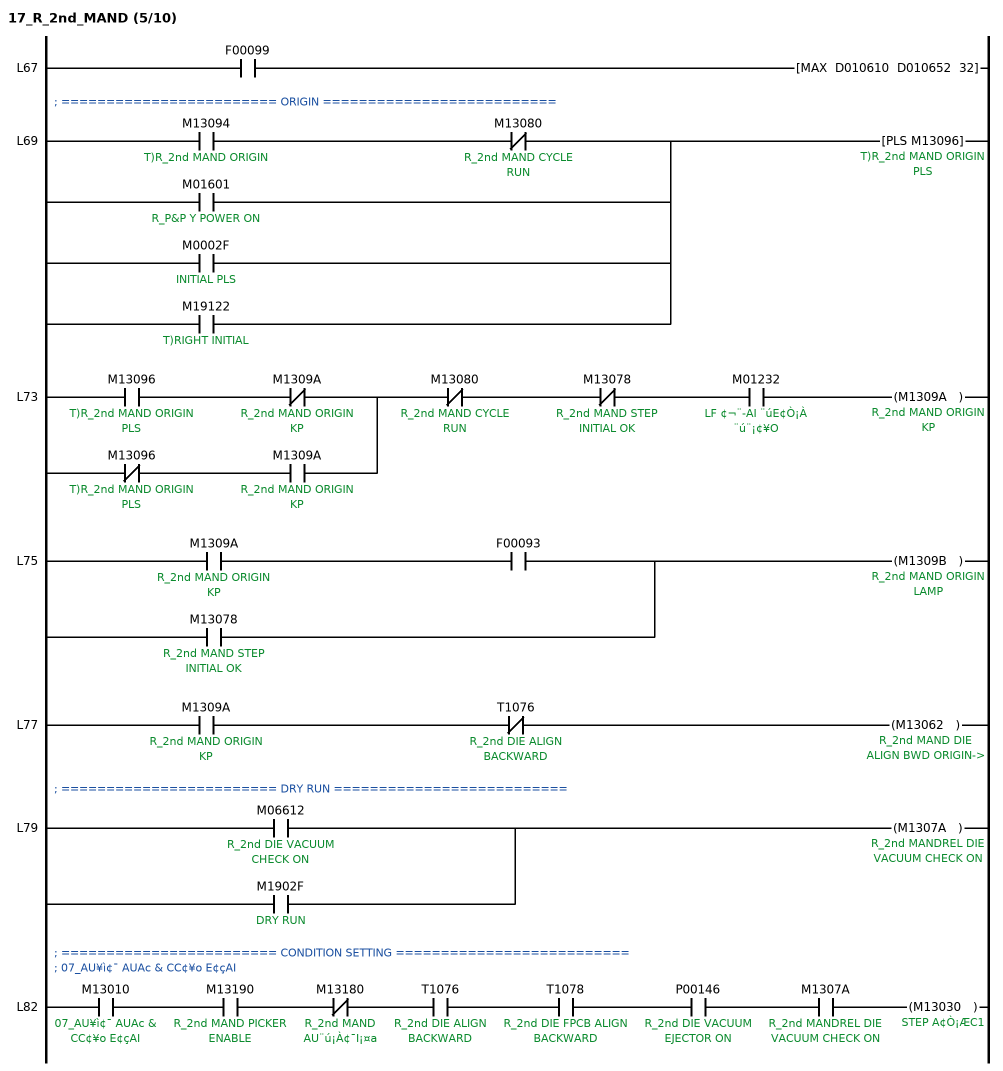
[picture p144: 17_R_2nd_MAND rungs L67-L82]
; L67
LOAD      F00099
MAX       D010610 D010652 32
// ======================== ORIGIN ==========================
; L69
LOAD      M13094	// T)R_2nd MAND ORIGIN
AND NOT   M13080	// R_2nd MAND CYCLE RUN
OR        M01601	// R_P&P Y POWER ON
OR        M0002F	// INITIAL PLS
OR        M19122	// T)RIGHT INITIAL
OUTP      M13096	// T)R_2nd MAND ORIGIN PLS
; L73
LOAD      M13096	// T)R_2nd MAND ORIGIN PLS
AND NOT   M1309A	// R_2nd MAND ORIGIN KP
LOAD NOT  M13096	// T)R_2nd MAND ORIGIN PLS
AND       M1309A	// R_2nd MAND ORIGIN KP
OR LOAD
AND NOT   M13080	// R_2nd MAND CYCLE RUN
AND NOT   M13078	// R_2nd MAND STEP INITIAL OK
AND       M01232	// LF ¢¬¨­AI ¨úE¢Ò¡À ¨ú¨¡¢¥O
OUT       M1309A	// R_2nd MAND ORIGIN KP
; L75
LOAD      M1309A	// R_2nd MAND ORIGIN KP
AND       F00093
OR        M13078	// R_2nd MAND STEP INITIAL OK
OUT       M1309B	// R_2nd MAND ORIGIN LAMP
; L77
LOAD      M1309A	// R_2nd MAND ORIGIN KP
AND NOT   T1076	// R_2nd DIE ALIGN BACKWARD
OUT       M13062	// R_2nd MAND DIE ALIGN BWD ORIGIN->
// ======================== DRY RUN ==========================
; L79
LOAD      M06612	// R_2nd DIE VACUUM CHECK ON
OR        M1902F	// DRY RUN
OUT       M1307A	// R_2nd MANDREL DIE VACUUM CHECK ON
// ======================== CONDITION SETTING ==========================
; L82
LOAD      M13010	// 07_AU¥ì¢¯ AUAc & CC¢¥o E¢çAI
AND       M13190	// R_2nd MAND PICKER ENABLE
AND NOT   M13180	// R_2nd MAND AU¨ú¡À¢¯I¡¤a
AND       T1076	// R_2nd DIE ALIGN BACKWARD
AND       T1078	// R_2nd DIE FPCB ALIGN BACKWARD
AND       P00146	// R_2nd DIE VACUUM EJECTOR ON
AND       M1307A	// R_2nd MANDREL DIE VACUUM CHECK ON
OUT       M13030	// STEP A¢Ò¡ÆC1
// output comment: 07_AU¥ì¢¯ AUAc & CC¢¥o E¢çAI

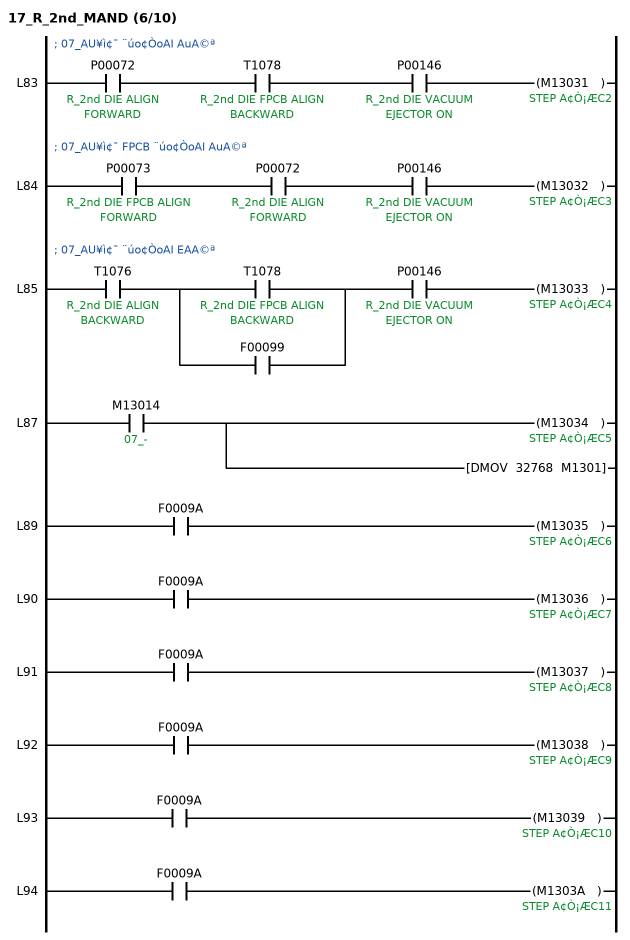
; L83
LOAD      P00072	// R_2nd DIE ALIGN FORWARD
AND       T1078	// R_2nd DIE FPCB ALIGN BACKWARD
AND       P00146	// R_2nd DIE VACUUM EJECTOR ON
OUT       M13031	// STEP A¢Ò¡ÆC2
// output comment: 07_AU¥ì¢¯ ¨úo¢ÒoAI AuA©ª
; L84
LOAD      P00073	// R_2nd DIE FPCB ALIGN FORWARD
AND       P00072	// R_2nd DIE ALIGN FORWARD
AND       P00146	// R_2nd DIE VACUUM EJECTOR ON
OUT       M13032	// STEP A¢Ò¡ÆC3
// output comment: 07_AU¥ì¢¯ FPCB ¨úo¢ÒoAI AuA©ª
; L85
LOAD      T1076	// R_2nd DIE ALIGN BACKWARD
LOAD      T1078	// R_2nd DIE FPCB ALIGN BACKWARD
OR        F00099
AND LOAD
AND       P00146	// R_2nd DIE VACUUM EJECTOR ON
OUT       M13033	// STEP A¢Ò¡ÆC4
// output comment: 07_AU¥ì¢¯ ¨úo¢ÒoAI EAA©ª
; L87
LOAD      M13014	// 07_-
OUT       M13034	// STEP A¢Ò¡ÆC5
DMOV      32768 M1301
; L89
LOAD      F0009A
OUT       M13035	// STEP A¢Ò¡ÆC6
; L90
LOAD      F0009A
OUT       M13036	// STEP A¢Ò¡ÆC7
; L91
LOAD      F0009A
OUT       M13037	// STEP A¢Ò¡ÆC8
; L92
LOAD      F0009A
OUT       M13038	// STEP A¢Ò¡ÆC9
; L93
LOAD      F0009A
OUT       M13039	// STEP A¢Ò¡ÆC10
; L94
LOAD      F0009A
OUT       M1303A	// STEP A¢Ò¡ÆC11

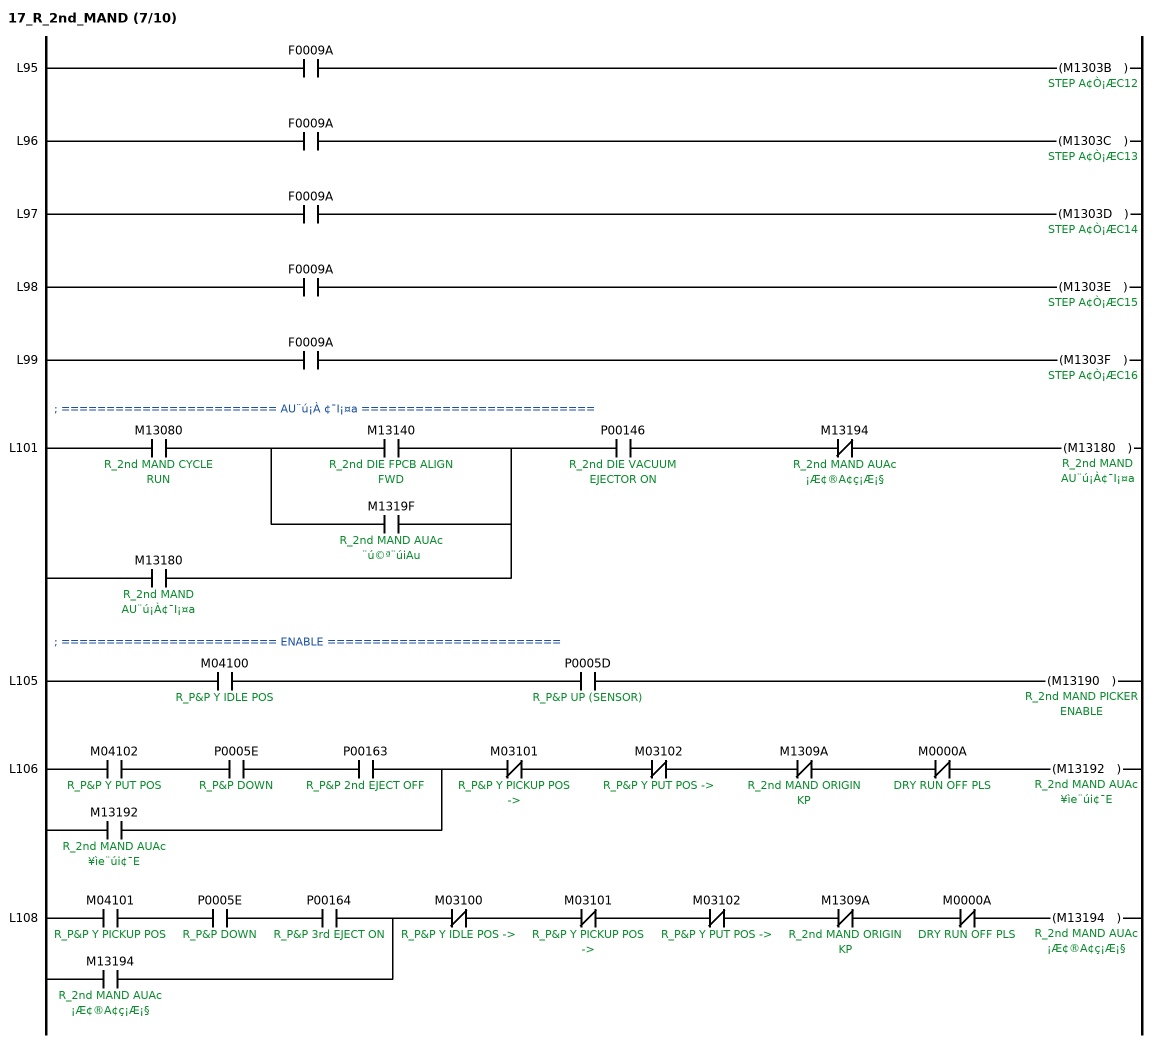
; L95
LOAD      F0009A
OUT       M1303B	// STEP A¢Ò¡ÆC12
; L96
LOAD      F0009A
OUT       M1303C	// STEP A¢Ò¡ÆC13
; L97
LOAD      F0009A
OUT       M1303D	// STEP A¢Ò¡ÆC14
; L98
LOAD      F0009A
OUT       M1303E	// STEP A¢Ò¡ÆC15
; L99
LOAD      F0009A
OUT       M1303F	// STEP A¢Ò¡ÆC16
// ======================== AU¨ú¡À ¢¯I¡¤a ==========================
; L101
LOAD      M13080	// R_2nd MAND CYCLE RUN
LOAD      M13140	// R_2nd DIE FPCB ALIGN FWD
OR        M1319F	// R_2nd MAND AUAc ¨ú©ª¨úiAu
AND LOAD
OR        M13180	// R_2nd MAND AU¨ú¡À¢¯I¡¤a
AND       P00146	// R_2nd DIE VACUUM EJECTOR ON
AND NOT   M13194	// R_2nd MAND AUAc ¡Æ¢®A¢ç¡Æ¡§
OUT       M13180	// R_2nd MAND AU¨ú¡À¢¯I¡¤a
// ======================== ENABLE ==========================
; L105
LOAD      M04100	// R_P&P Y IDLE POS
AND       P0005D	// R_P&P UP (SENSOR)
OUT       M13190	// R_2nd MAND PICKER ENABLE
; L106
LOAD      M04102	// R_P&P Y PUT POS
AND       P0005E	// R_P&P DOWN
AND       P00163	// R_P&P 2nd EJECT OFF
OR        M13192	// R_2nd MAND AUAc ¥ìe¨úi¢¯E
AND NOT   M03101	// R_P&P Y PICKUP POS ->
AND NOT   M03102	// R_P&P Y PUT POS ->
AND NOT   M1309A	// R_2nd MAND ORIGIN KP
AND NOT   M0000A	// DRY RUN OFF PLS
OUT       M13192	// R_2nd MAND AUAc ¥ìe¨úi¢¯E
; L108
LOAD      M04101	// R_P&P Y PICKUP POS
AND       P0005E	// R_P&P DOWN
AND       P00164	// R_P&P 3rd EJECT ON
OR        M13194	// R_2nd MAND AUAc ¡Æ¢®A¢ç¡Æ¡§
AND NOT   M03100	// R_P&P Y IDLE POS ->
AND NOT   M03101	// R_P&P Y PICKUP POS ->
AND NOT   M03102	// R_P&P Y PUT POS ->
AND NOT   M1309A	// R_2nd MAND ORIGIN KP
AND NOT   M0000A	// DRY RUN OFF PLS
OUT       M13194	// R_2nd MAND AUAc ¡Æ¢®A¢ç¡Æ¡§

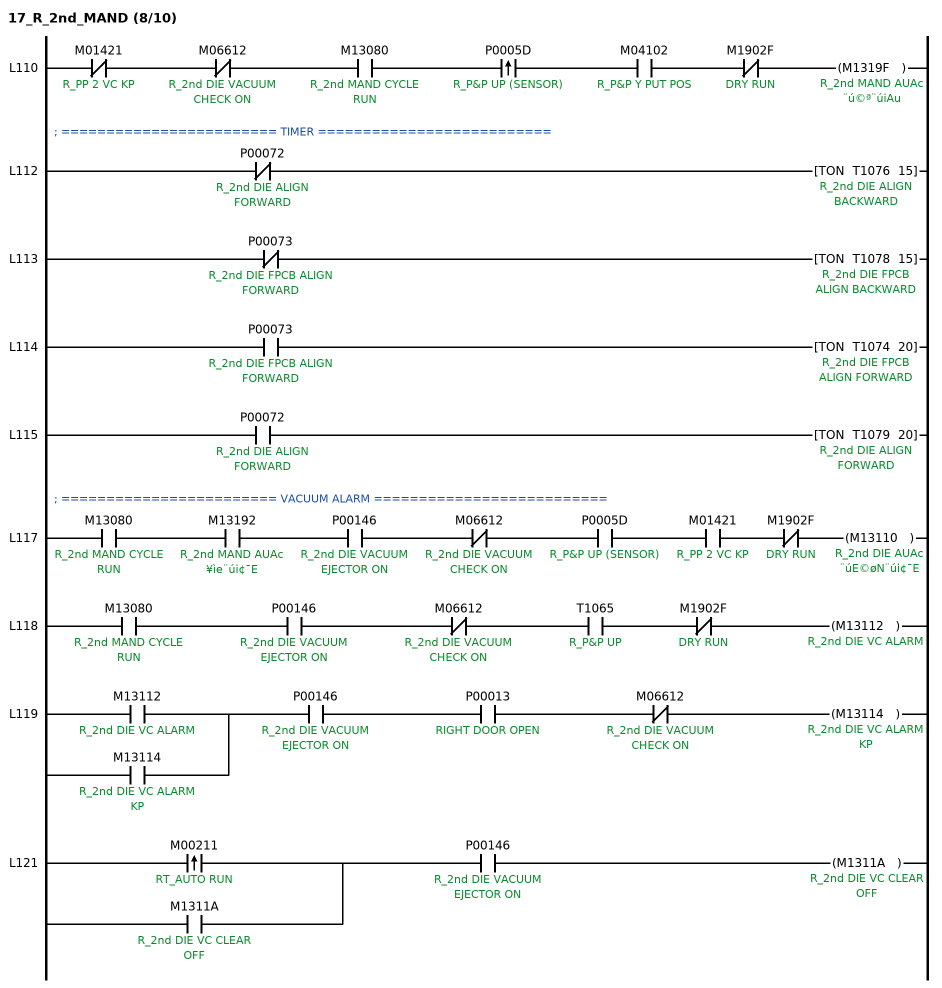
; L110
LOAD NOT  M01421	// R_PP 2 VC KP
AND NOT   M06612	// R_2nd DIE VACUUM CHECK ON
AND       M13080	// R_2nd MAND CYCLE RUN
ANDP      P0005D	// R_P&P UP (SENSOR)
AND       M04102	// R_P&P Y PUT POS
AND NOT   M1902F	// DRY RUN
OUT       M1319F	// R_2nd MAND AUAc ¨ú©ª¨úiAu
// ======================== TIMER ==========================
; L112
LOAD NOT  P00072	// R_2nd DIE ALIGN FORWARD
TON       T1076 15	// R_2nd DIE ALIGN BACKWARD
; L113
LOAD NOT  P00073	// R_2nd DIE FPCB ALIGN FORWARD
TON       T1078 15	// R_2nd DIE FPCB ALIGN BACKWARD
; L114
LOAD      P00073	// R_2nd DIE FPCB ALIGN FORWARD
TON       T1074 20	// R_2nd DIE FPCB ALIGN FORWARD
; L115
LOAD      P00072	// R_2nd DIE ALIGN FORWARD
TON       T1079 20	// R_2nd DIE ALIGN FORWARD
// ======================== VACUUM ALARM ==========================
; L117
LOAD      M13080	// R_2nd MAND CYCLE RUN
AND       M13192	// R_2nd MAND AUAc ¥ìe¨úi¢¯E
AND       P00146	// R_2nd DIE VACUUM EJECTOR ON
AND NOT   M06612	// R_2nd DIE VACUUM CHECK ON
AND       P0005D	// R_P&P UP (SENSOR)
AND       M01421	// R_PP 2 VC KP
AND NOT   M1902F	// DRY RUN
OUT       M13110	// R_2nd DIE AUAc ¨úE©øN¨úi¢¯E
; L118
LOAD      M13080	// R_2nd MAND CYCLE RUN
AND       P00146	// R_2nd DIE VACUUM EJECTOR ON
AND NOT   M06612	// R_2nd DIE VACUUM CHECK ON
AND       T1065	// R_P&P UP
AND NOT   M1902F	// DRY RUN
OUT       M13112	// R_2nd DIE VC ALARM
; L119
LOAD      M13112	// R_2nd DIE VC ALARM
OR        M13114	// R_2nd DIE VC ALARM KP
AND       P00146	// R_2nd DIE VACUUM EJECTOR ON
AND       P00013	// RIGHT DOOR OPEN
AND NOT   M06612	// R_2nd DIE VACUUM CHECK ON
OUT       M13114	// R_2nd DIE VC ALARM KP
; L121
LOADP     M00211	// RT_AUTO RUN
OR        M1311A	// R_2nd DIE VC CLEAR OFF
AND       P00146	// R_2nd DIE VACUUM EJECTOR ON
OUT       M1311A	// R_2nd DIE VC CLEAR OFF

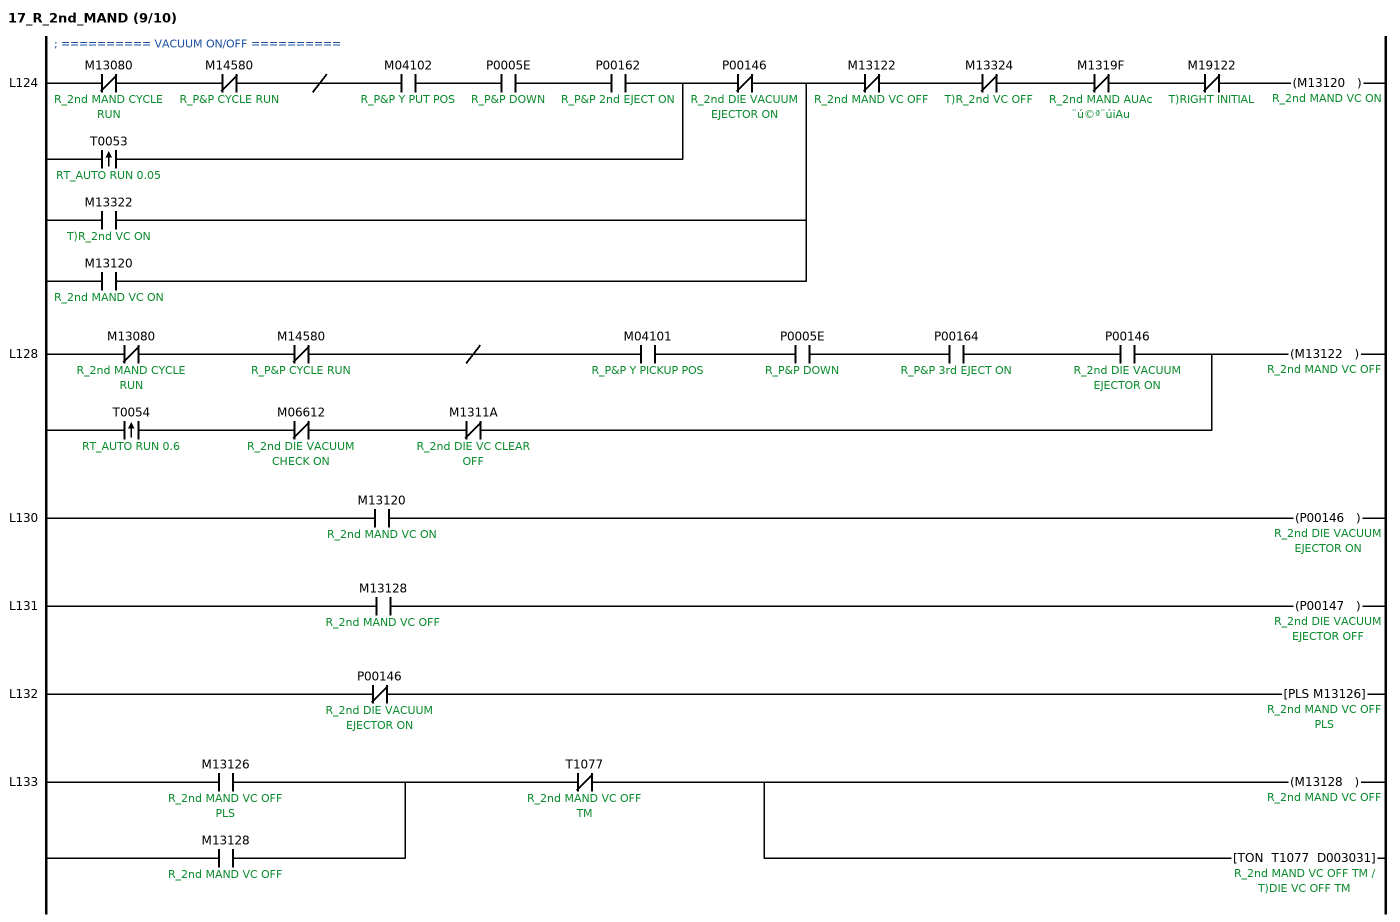
// ========== VACUUM ON/OFF ==========
; L124
LOAD NOT  M13080	// R_2nd MAND CYCLE RUN
AND NOT   M14580	// R_P&P CYCLE RUN
NOT
AND       M04102	// R_P&P Y PUT POS
AND       P0005E	// R_P&P DOWN
AND       P00162	// R_P&P 2nd EJECT ON
ORP       T0053	// RT_AUTO RUN 0.05
AND NOT   P00146	// R_2nd DIE VACUUM EJECTOR ON
OR        M13322	// T)R_2nd VC ON
OR        M13120	// R_2nd MAND VC ON
AND NOT   M13122	// R_2nd MAND VC OFF
AND NOT   M13324	// T)R_2nd VC OFF
AND NOT   M1319F	// R_2nd MAND AUAc ¨ú©ª¨úiAu
AND NOT   M19122	// T)RIGHT INITIAL
OUT       M13120	// R_2nd MAND VC ON
; L128
LOAD NOT  M13080	// R_2nd MAND CYCLE RUN
AND NOT   M14580	// R_P&P CYCLE RUN
NOT
AND       M04101	// R_P&P Y PICKUP POS
AND       P0005E	// R_P&P DOWN
AND       P00164	// R_P&P 3rd EJECT ON
AND       P00146	// R_2nd DIE VACUUM EJECTOR ON
LOADP     T0054	// RT_AUTO RUN 0.6
AND NOT   M06612	// R_2nd DIE VACUUM CHECK ON
AND NOT   M1311A	// R_2nd DIE VC CLEAR OFF
OR LOAD
OUT       M13122	// R_2nd MAND VC OFF
; L130
LOAD      M13120	// R_2nd MAND VC ON
OUT       P00146	// R_2nd DIE VACUUM EJECTOR ON
; L131
LOAD      M13128	// R_2nd MAND VC OFF
OUT       P00147	// R_2nd DIE VACUUM EJECTOR OFF
; L132
LOAD NOT  P00146	// R_2nd DIE VACUUM EJECTOR ON
OUTP      M13126	// R_2nd MAND VC OFF PLS
; L133
LOAD      M13126	// R_2nd MAND VC OFF PLS
OR        M13128	// R_2nd MAND VC OFF
AND NOT   T1077	// R_2nd MAND VC OFF TM
OUT       M13128	// R_2nd MAND VC OFF
TON       T1077 D003031	// R_2nd MAND VC OFF TM / T)DIE VC OFF TM

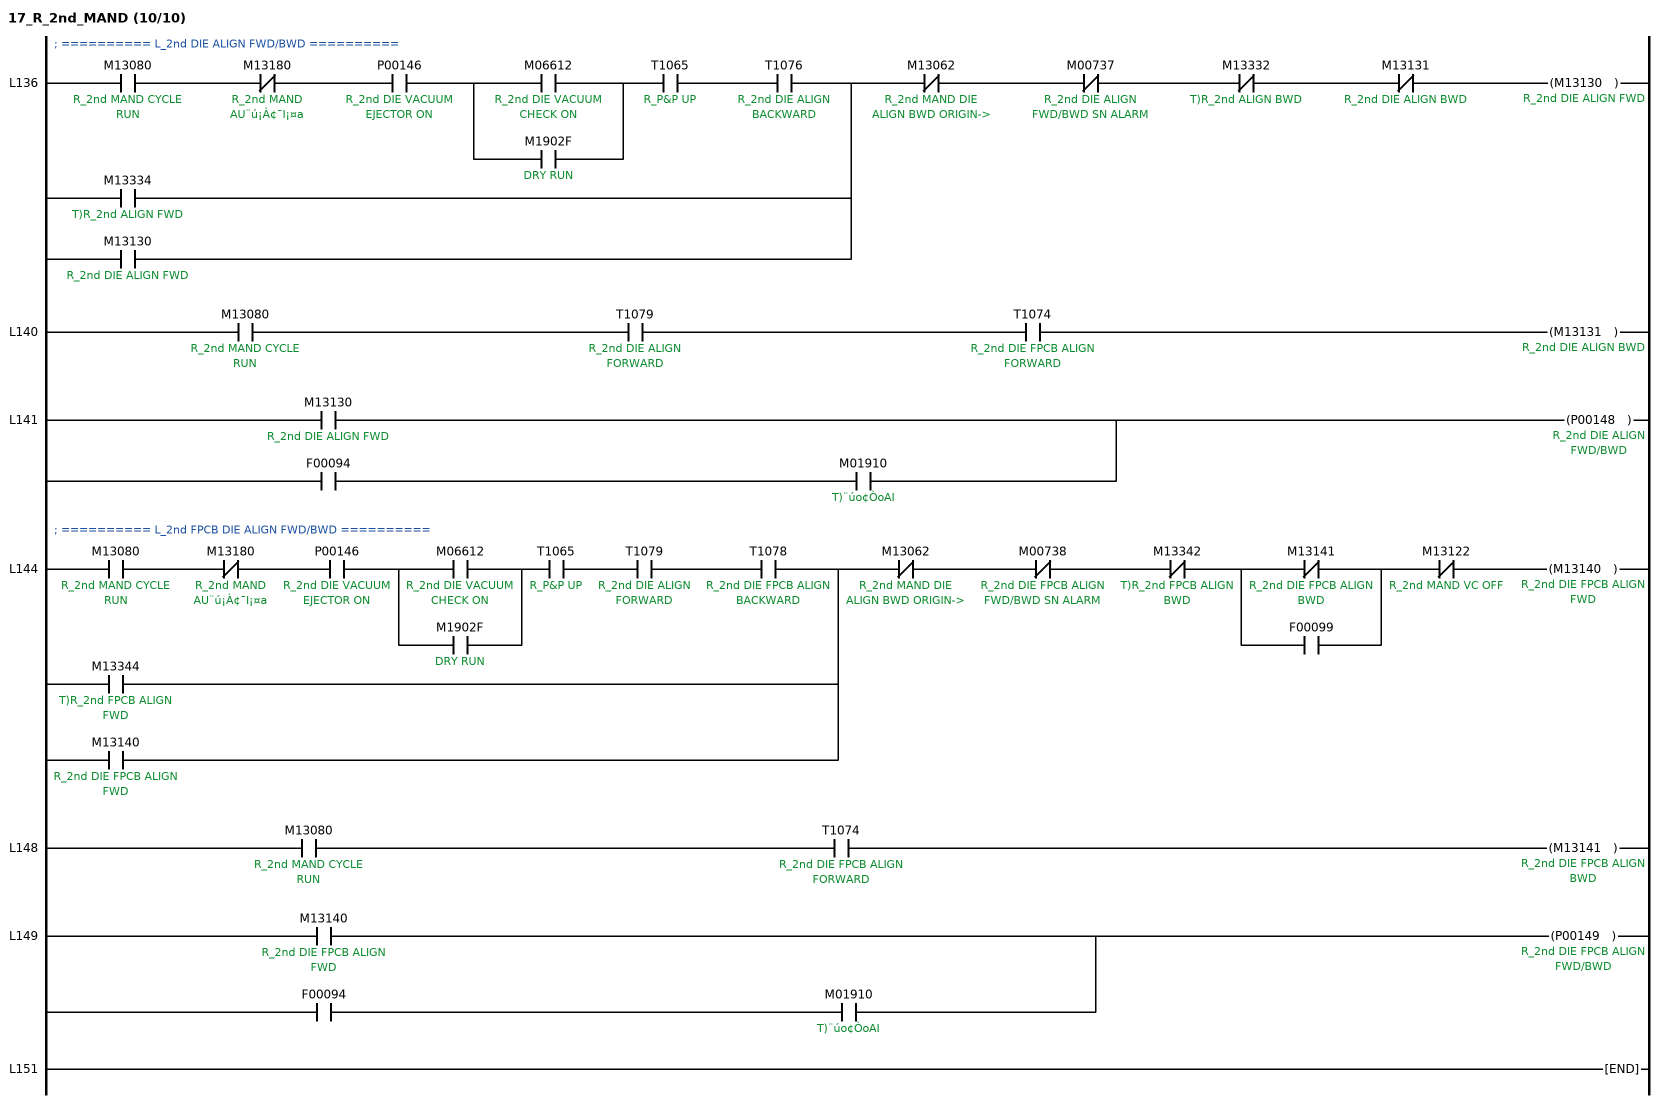
// ========== L_2nd DIE ALIGN FWD/BWD ==========
; L136
LOAD      M13080	// R_2nd MAND CYCLE RUN
AND NOT   M13180	// R_2nd MAND AU¨ú¡À¢¯I¡¤a
AND       P00146	// R_2nd DIE VACUUM EJECTOR ON
LOAD      M06612	// R_2nd DIE VACUUM CHECK ON
OR        M1902F	// DRY RUN
AND LOAD
AND       T1065	// R_P&P UP
AND       T1076	// R_2nd DIE ALIGN BACKWARD
OR        M13334	// T)R_2nd ALIGN FWD
OR        M13130	// R_2nd DIE ALIGN FWD
AND NOT   M13062	// R_2nd MAND DIE ALIGN BWD ORIGIN->
AND NOT   M00737	// R_2nd DIE ALIGN FWD/BWD SN ALARM
AND NOT   M13332	// T)R_2nd ALIGN BWD
AND NOT   M13131	// R_2nd DIE ALIGN BWD
OUT       M13130	// R_2nd DIE ALIGN FWD
; L140
LOAD      M13080	// R_2nd MAND CYCLE RUN
AND       T1079	// R_2nd DIE ALIGN FORWARD
AND       T1074	// R_2nd DIE FPCB ALIGN FORWARD
OUT       M13131	// R_2nd DIE ALIGN BWD
; L141
LOAD      M13130	// R_2nd DIE ALIGN FWD
LOAD      F00094
AND       M01910	// T)¨úo¢ÒoAI
OR LOAD
OUT       P00148	// R_2nd DIE ALIGN FWD/BWD
// ========== L_2nd FPCB DIE ALIGN FWD/BWD ==========
; L144
LOAD      M13080	// R_2nd MAND CYCLE RUN
AND NOT   M13180	// R_2nd MAND AU¨ú¡À¢¯I¡¤a
AND       P00146	// R_2nd DIE VACUUM EJECTOR ON
LOAD      M06612	// R_2nd DIE VACUUM CHECK ON
OR        M1902F	// DRY RUN
AND LOAD
AND       T1065	// R_P&P UP
AND       T1079	// R_2nd DIE ALIGN FORWARD
AND       T1078	// R_2nd DIE FPCB ALIGN BACKWARD
OR        M13344	// T)R_2nd FPCB ALIGN FWD
OR        M13140	// R_2nd DIE FPCB ALIGN FWD
AND NOT   M13062	// R_2nd MAND DIE ALIGN BWD ORIGIN->
AND NOT   M00738	// R_2nd DIE FPCB ALIGN FWD/BWD SN ALARM
AND NOT   M13342	// T)R_2nd FPCB ALIGN BWD
LOAD NOT  M13141	// R_2nd DIE FPCB ALIGN BWD
OR        F00099
AND LOAD
AND NOT   M13122	// R_2nd MAND VC OFF
OUT       M13140	// R_2nd DIE FPCB ALIGN FWD
; L148
LOAD      M13080	// R_2nd MAND CYCLE RUN
AND       T1074	// R_2nd DIE FPCB ALIGN FORWARD
OUT       M13141	// R_2nd DIE FPCB ALIGN BWD
; L149
LOAD      M13140	// R_2nd DIE FPCB ALIGN FWD
LOAD      F00094
AND       M01910	// T)¨úo¢ÒoAI
OR LOAD
OUT       P00149	// R_2nd DIE FPCB ALIGN FWD/BWD
; L151
END

PROGRAM 18_R_3rd_MAND (task: ¨ö¨¬A¥ì CA¡¤I¡¾¡¿¡¤¡Í)

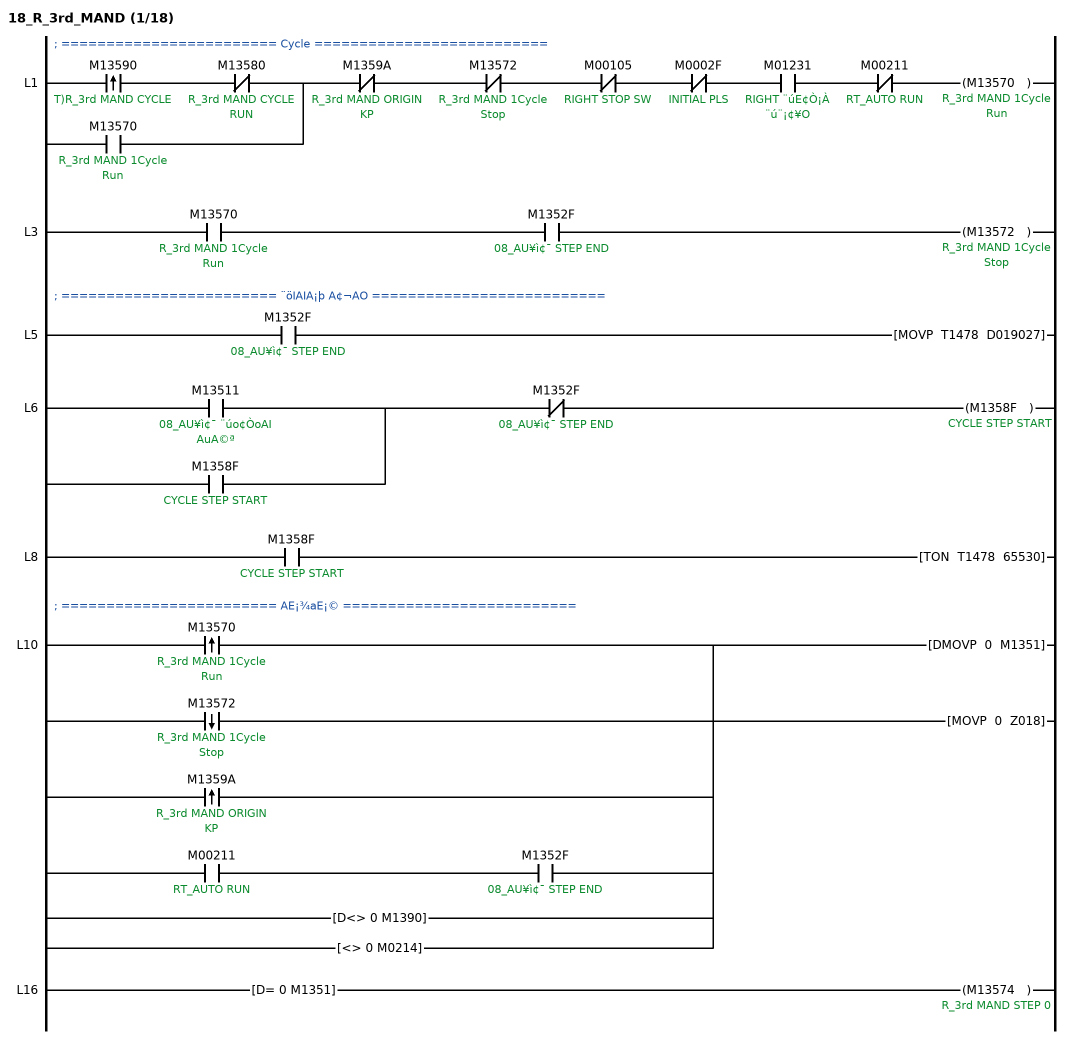
// ======================== Cycle ==========================
; L1
LOADP     M13590	// T)R_3rd MAND CYCLE
AND NOT   M13580	// R_3rd MAND CYCLE RUN
OR        M13570	// R_3rd MAND 1Cycle Run
AND NOT   M1359A	// R_3rd MAND ORIGIN KP
AND NOT   M13572	// R_3rd MAND 1Cycle Stop
AND NOT   M00105	// RIGHT STOP SW
AND NOT   M0002F	// INITIAL PLS
AND       M01231	// RIGHT ¨úE¢Ò¡À ¨ú¨¡¢¥O
AND NOT   M00211	// RT_AUTO RUN
OUT       M13570	// R_3rd MAND 1Cycle Run
; L3
LOAD      M13570	// R_3rd MAND 1Cycle Run
AND       M1352F	// 08_AU¥ì¢¯ STEP END
OUT       M13572	// R_3rd MAND 1Cycle Stop
// ======================== ¨öIAIA¡þ A¢¬AO ==========================
; L5
LOAD      M1352F	// 08_AU¥ì¢¯ STEP END
MOVP      T1478 D019027
; L6
LOAD      M13511	// 08_AU¥ì¢¯ ¨úo¢ÒoAI AuA©ª
OR        M1358F	// CYCLE STEP START
AND NOT   M1352F	// 08_AU¥ì¢¯ STEP END
OUT       M1358F	// CYCLE STEP START
; L8
LOAD      M1358F	// CYCLE STEP START
TON       T1478 65530
// ======================== AE¡¾aE¡© ==========================
; L10
LOADP     M13570	// R_3rd MAND 1Cycle Run
ORN       M13572	// R_3rd MAND 1Cycle Stop
ORP       M1359A	// R_3rd MAND ORIGIN KP
LOAD      M00211	// RT_AUTO RUN
AND       M1352F	// 08_AU¥ì¢¯ STEP END
OR LOAD
ORD<>     0 M1390
OR<>      0 M0214
DMOVP     0 M1351
MOVP      0 Z018
; L16
LOADD=    0 M1351
OUT       M13574	// R_3rd MAND STEP 0

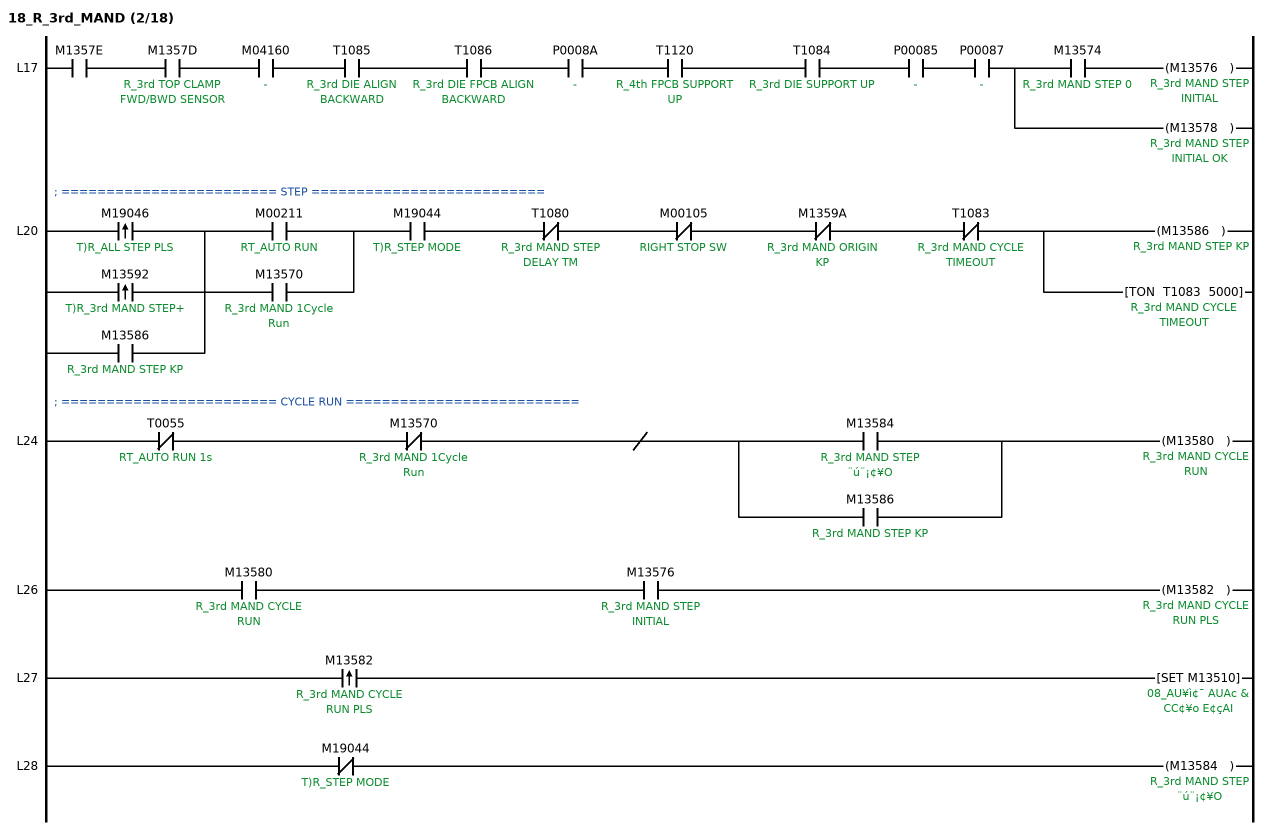
; L17
LOAD      M1357E
AND       M1357D	// R_3rd TOP CLAMP FWD/BWD SENSOR
AND       M04160	// -
AND       T1085	// R_3rd DIE ALIGN BACKWARD
AND       T1086	// R_3rd DIE FPCB ALIGN BACKWARD
AND       P0008A	// -
AND       T1120	// R_4th FPCB SUPPORT UP
AND       T1084	// R_3rd DIE SUPPORT UP
AND       P00085	// -
AND       P00087	// -
MPUSH
AND       M13574	// R_3rd MAND STEP 0
OUT       M13576	// R_3rd MAND STEP INITIAL
MPOP
OUT       M13578	// R_3rd MAND STEP INITIAL OK
// ======================== STEP ==========================
; L20
LOADP     M19046	// T)R_ALL STEP PLS
ORP       M13592	// T)R_3rd MAND STEP+
OR        M13586	// R_3rd MAND STEP KP
LOAD      M00211	// RT_AUTO RUN
OR        M13570	// R_3rd MAND 1Cycle Run
AND LOAD
AND       M19044	// T)R_STEP MODE
AND NOT   T1080	// R_3rd MAND STEP DELAY TM
AND NOT   M00105	// RIGHT STOP SW
AND NOT   M1359A	// R_3rd MAND ORIGIN KP
AND NOT   T1083	// R_3rd MAND CYCLE TIMEOUT
OUT       M13586	// R_3rd MAND STEP KP
TON       T1083 5000	// R_3rd MAND CYCLE TIMEOUT
// ======================== CYCLE RUN ==========================
; L24
LOAD NOT  T0055	// RT_AUTO RUN 1s
AND NOT   M13570	// R_3rd MAND 1Cycle Run
NOT
LOAD      M13584	// R_3rd MAND STEP ¨ú¨¡¢¥O
OR        M13586	// R_3rd MAND STEP KP
AND LOAD
OUT       M13580	// R_3rd MAND CYCLE RUN
; L26
LOAD      M13580	// R_3rd MAND CYCLE RUN
AND       M13576	// R_3rd MAND STEP INITIAL
OUT       M13582	// R_3rd MAND CYCLE RUN PLS
; L27
LOADP     M13582	// R_3rd MAND CYCLE RUN PLS
SET       M13510	// 08_AU¥ì¢¯ AUAc & CC¢¥o E¢çAI
; L28
LOAD NOT  M19044	// T)R_STEP MODE
OUT       M13584	// R_3rd MAND STEP ¨ú¨¡¢¥O

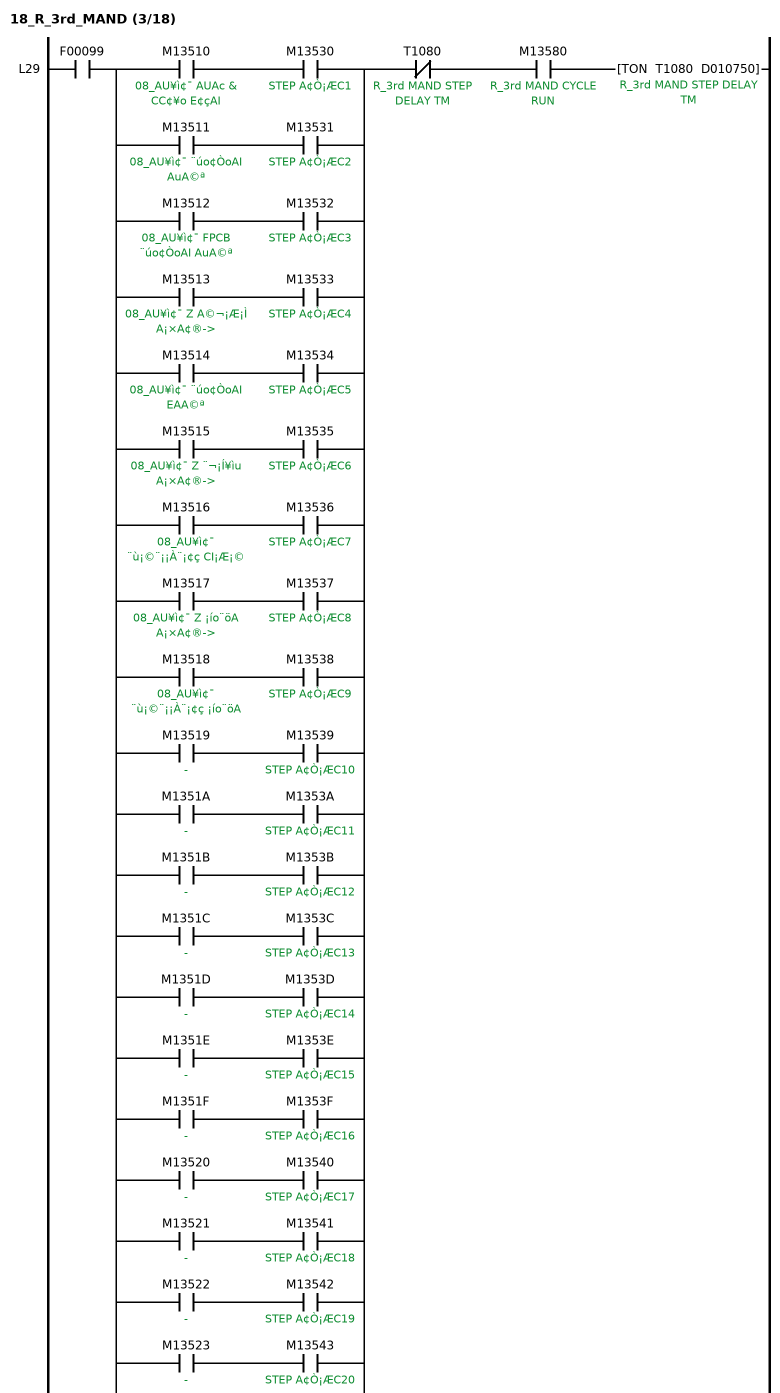

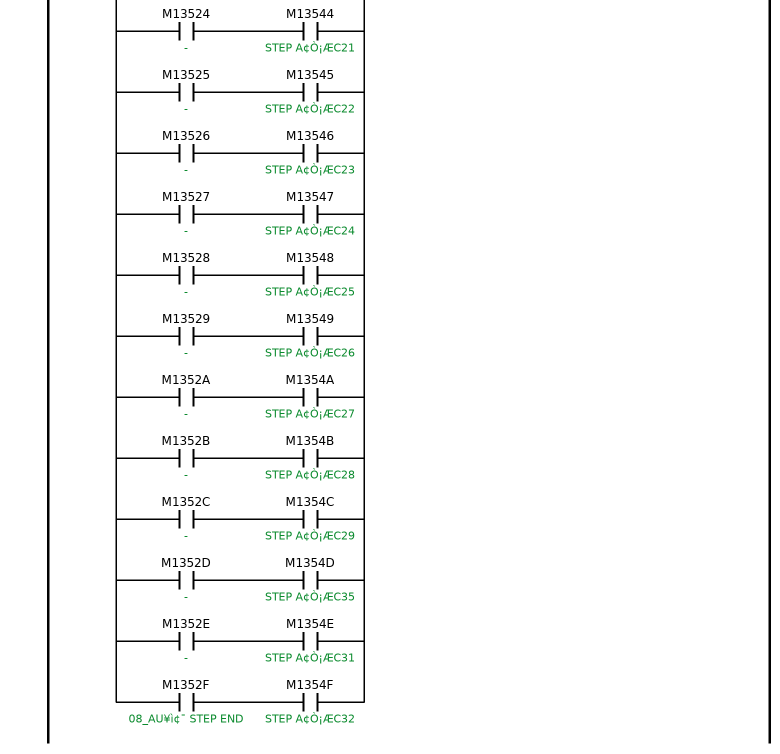
; L29
LOAD      F00099
LOAD      M13510	// 08_AU¥ì¢¯ AUAc & CC¢¥o E¢çAI
AND       M13530	// STEP A¢Ò¡ÆC1
LOAD      M13511	// 08_AU¥ì¢¯ ¨úo¢ÒoAI AuA©ª
AND       M13531	// STEP A¢Ò¡ÆC2
OR LOAD
LOAD      M13512	// 08_AU¥ì¢¯ FPCB ¨úo¢ÒoAI AuA©ª
AND       M13532	// STEP A¢Ò¡ÆC3
OR LOAD
LOAD      M13513	// 08_AU¥ì¢¯ Z A©¬¡Æ¡Ì A¡×A¢®->
AND       M13533	// STEP A¢Ò¡ÆC4
OR LOAD
LOAD      M13514	// 08_AU¥ì¢¯ ¨úo¢ÒoAI EAA©ª
AND       M13534	// STEP A¢Ò¡ÆC5
OR LOAD
LOAD      M13515	// 08_AU¥ì¢¯ Z ¨¬¡Í¥ìu A¡×A¢®->
AND       M13535	// STEP A¢Ò¡ÆC6
OR LOAD
LOAD      M13516	// 08_AU¥ì¢¯ ¨ù¡©¨¡¡À¨¡¢ç CI¡Æ¡©
AND       M13536	// STEP A¢Ò¡ÆC7
OR LOAD
LOAD      M13517	// 08_AU¥ì¢¯ Z ¡ío¨öA A¡×A¢®->
AND       M13537	// STEP A¢Ò¡ÆC8
OR LOAD
LOAD      M13518	// 08_AU¥ì¢¯ ¨ù¡©¨¡¡À¨¡¢ç ¡ío¨öA
AND       M13538	// STEP A¢Ò¡ÆC9
OR LOAD
LOAD      M13519	// -
AND       M13539	// STEP A¢Ò¡ÆC10
OR LOAD
LOAD      M1351A	// -
AND       M1353A	// STEP A¢Ò¡ÆC11
OR LOAD
LOAD      M1351B	// -
AND       M1353B	// STEP A¢Ò¡ÆC12
OR LOAD
LOAD      M1351C	// -
AND       M1353C	// STEP A¢Ò¡ÆC13
OR LOAD
LOAD      M1351D	// -
AND       M1353D	// STEP A¢Ò¡ÆC14
OR LOAD
LOAD      M1351E	// -
AND       M1353E	// STEP A¢Ò¡ÆC15
OR LOAD
LOAD      M1351F	// -
AND       M1353F	// STEP A¢Ò¡ÆC16
OR LOAD
LOAD      M13520	// -
AND       M13540	// STEP A¢Ò¡ÆC17
OR LOAD
LOAD      M13521	// -
AND       M13541	// STEP A¢Ò¡ÆC18
OR LOAD
LOAD      M13522	// -
AND       M13542	// STEP A¢Ò¡ÆC19
OR LOAD
LOAD      M13523	// -
AND       M13543	// STEP A¢Ò¡ÆC20
OR LOAD
LOAD      M13524	// -
AND       M13544	// STEP A¢Ò¡ÆC21
OR LOAD
LOAD      M13525	// -
AND       M13545	// STEP A¢Ò¡ÆC22
OR LOAD
LOAD      M13526	// -
AND       M13546	// STEP A¢Ò¡ÆC23
OR LOAD
LOAD      M13527	// -
AND       M13547	// STEP A¢Ò¡ÆC24
OR LOAD
LOAD      M13528	// -
AND       M13548	// STEP A¢Ò¡ÆC25
OR LOAD
LOAD      M13529	// -
AND       M13549	// STEP A¢Ò¡ÆC26
OR LOAD
LOAD      M1352A	// -
AND       M1354A	// STEP A¢Ò¡ÆC27
OR LOAD
LOAD      M1352B	// -
AND       M1354B	// STEP A¢Ò¡ÆC28
OR LOAD
LOAD      M1352C	// -
AND       M1354C	// STEP A¢Ò¡ÆC29
OR LOAD
LOAD      M1352D	// -
AND       M1354D	// STEP A¢Ò¡ÆC35
OR LOAD
LOAD      M1352E	// -
AND       M1354E	// STEP A¢Ò¡ÆC31
OR LOAD
LOAD      M1352F	// 08_AU¥ì¢¯ STEP END
AND       M1354F	// STEP A¢Ò¡ÆC32
OR LOAD
AND LOAD
AND NOT   T1080	// R_3rd MAND STEP DELAY TM
AND       M13580	// R_3rd MAND CYCLE RUN
TON       T1080 D010750	// R_3rd MAND STEP DELAY TM

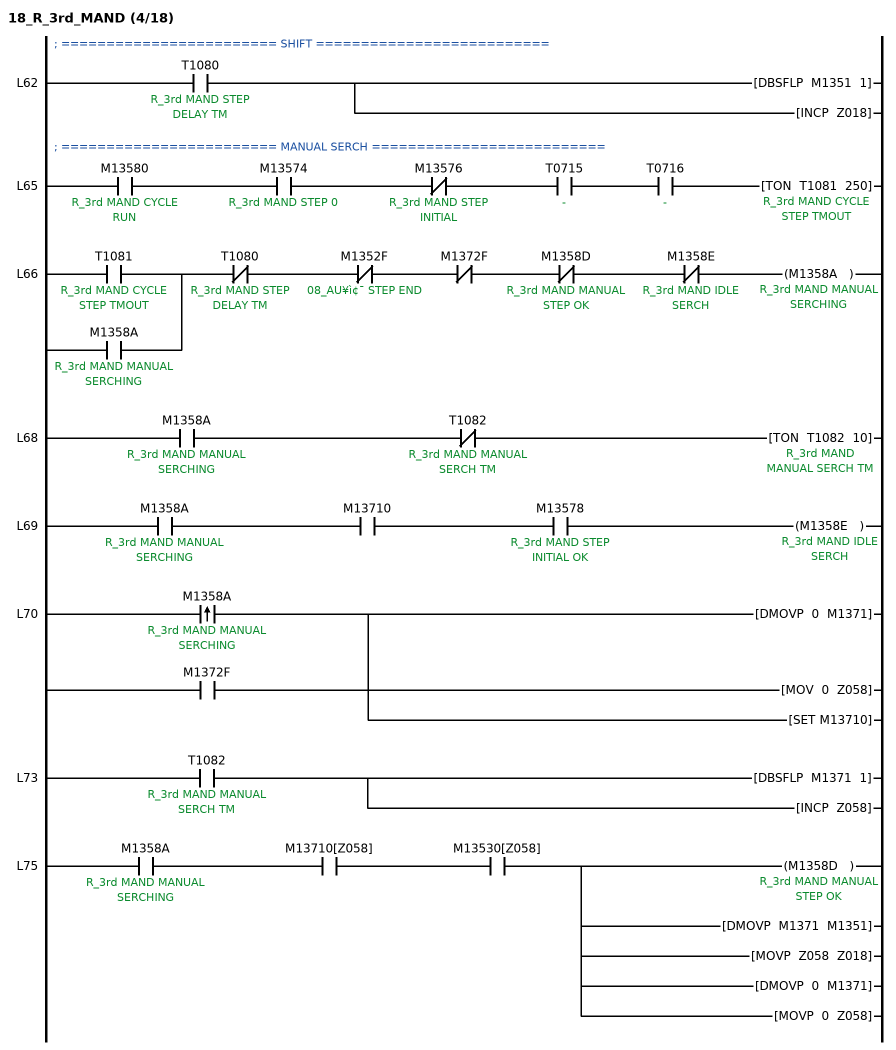
// ======================== SHIFT ==========================
; L62
LOAD      T1080	// R_3rd MAND STEP DELAY TM
DBSFLP    M1351 1
INCP      Z018
// ======================== MANUAL SERCH ==========================
; L65
LOAD      M13580	// R_3rd MAND CYCLE RUN
AND       M13574	// R_3rd MAND STEP 0
AND NOT   M13576	// R_3rd MAND STEP INITIAL
AND       T0715	// -
AND       T0716	// -
TON       T1081 250	// R_3rd MAND CYCLE STEP TMOUT
; L66
LOAD      T1081	// R_3rd MAND CYCLE STEP TMOUT
OR        M1358A	// R_3rd MAND MANUAL SERCHING
AND NOT   T1080	// R_3rd MAND STEP DELAY TM
AND NOT   M1352F	// 08_AU¥ì¢¯ STEP END
AND NOT   M1372F
AND NOT   M1358D	// R_3rd MAND MANUAL STEP OK
AND NOT   M1358E	// R_3rd MAND IDLE SERCH
OUT       M1358A	// R_3rd MAND MANUAL SERCHING
; L68
LOAD      M1358A	// R_3rd MAND MANUAL SERCHING
AND NOT   T1082	// R_3rd MAND MANUAL SERCH TM
TON       T1082 10	// R_3rd MAND MANUAL SERCH TM
; L69
LOAD      M1358A	// R_3rd MAND MANUAL SERCHING
AND       M13710
AND       M13578	// R_3rd MAND STEP INITIAL OK
OUT       M1358E	// R_3rd MAND IDLE SERCH
; L70
LOADP     M1358A	// R_3rd MAND MANUAL SERCHING
OR        M1372F
DMOVP     0 M1371
MOV       0 Z058
SET       M13710
; L73
LOAD      T1082	// R_3rd MAND MANUAL SERCH TM
DBSFLP    M1371 1
INCP      Z058
; L75
LOAD      M1358A	// R_3rd MAND MANUAL SERCHING
AND       M13710[Z058]
AND       M13530[Z058]
OUT       M1358D	// R_3rd MAND MANUAL STEP OK
DMOVP     M1371 M1351
MOVP      Z058 Z018
DMOVP     0 M1371
MOVP      0 Z058

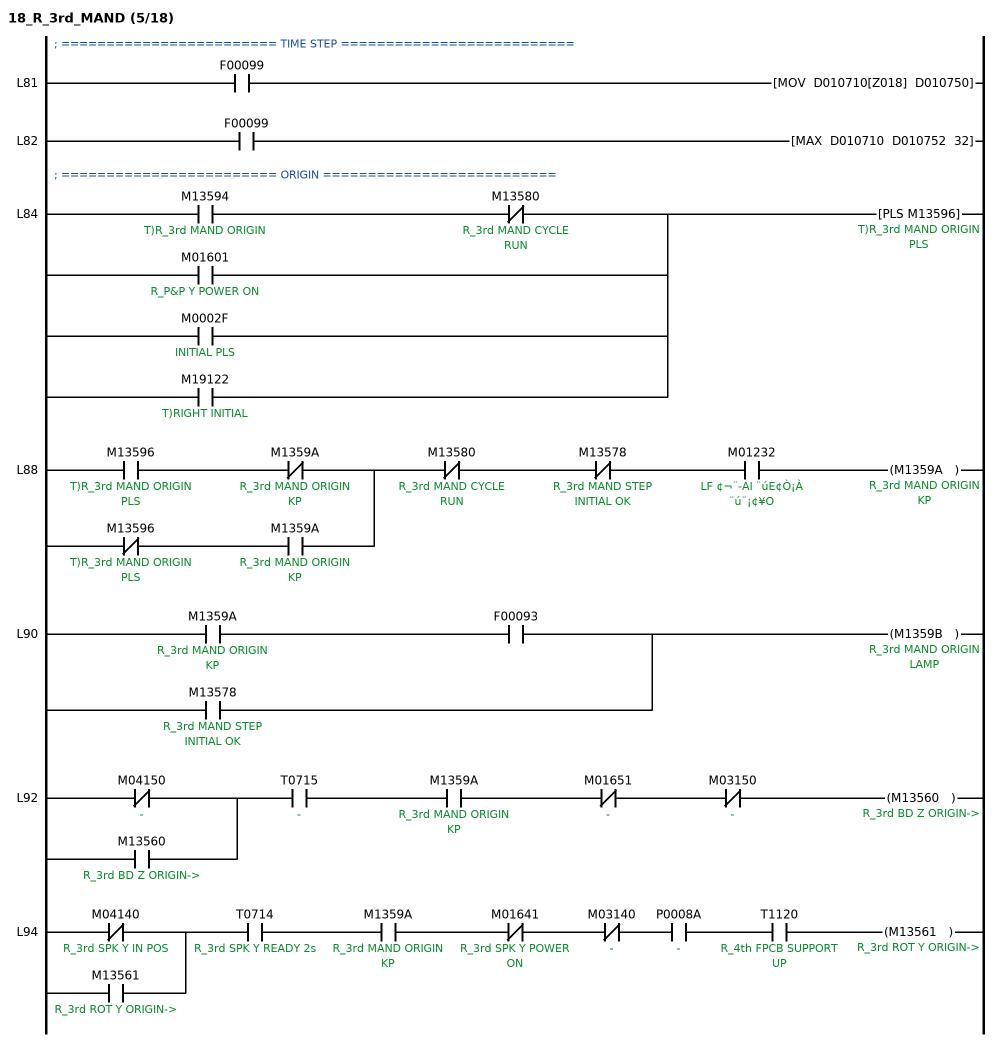
// ======================== TIME STEP ==========================
; L81
LOAD      F00099
MOV       D010710[Z018] D010750
; L82
LOAD      F00099
MAX       D010710 D010752 32
// ======================== ORIGIN ==========================
; L84
LOAD      M13594	// T)R_3rd MAND ORIGIN
AND NOT   M13580	// R_3rd MAND CYCLE RUN
OR        M01601	// R_P&P Y POWER ON
OR        M0002F	// INITIAL PLS
OR        M19122	// T)RIGHT INITIAL
OUTP      M13596	// T)R_3rd MAND ORIGIN PLS
; L88
LOAD      M13596	// T)R_3rd MAND ORIGIN PLS
AND NOT   M1359A	// R_3rd MAND ORIGIN KP
LOAD NOT  M13596	// T)R_3rd MAND ORIGIN PLS
AND       M1359A	// R_3rd MAND ORIGIN KP
OR LOAD
AND NOT   M13580	// R_3rd MAND CYCLE RUN
AND NOT   M13578	// R_3rd MAND STEP INITIAL OK
AND       M01232	// LF ¢¬¨­AI ¨úE¢Ò¡À ¨ú¨¡¢¥O
OUT       M1359A	// R_3rd MAND ORIGIN KP
; L90
LOAD      M1359A	// R_3rd MAND ORIGIN KP
AND       F00093
OR        M13578	// R_3rd MAND STEP INITIAL OK
OUT       M1359B	// R_3rd MAND ORIGIN LAMP
; L92
LOAD NOT  M04150	// -
OR        M13560	// R_3rd BD Z ORIGIN->
AND       T0715	// -
AND       M1359A	// R_3rd MAND ORIGIN KP
AND NOT   M01651	// -
AND NOT   M03150	// -
OUT       M13560	// R_3rd BD Z ORIGIN->
; L94
LOAD NOT  M04140	// R_3rd SPK Y IN POS
OR        M13561	// R_3rd ROT Y ORIGIN->
AND       T0714	// R_3rd SPK Y READY 2s
AND       M1359A	// R_3rd MAND ORIGIN KP
AND NOT   M01641	// R_3rd SPK Y POWER ON
AND NOT   M03140	// -
AND       P0008A	// -
AND       T1120	// R_4th FPCB SUPPORT UP
OUT       M13561	// R_3rd ROT Y ORIGIN->

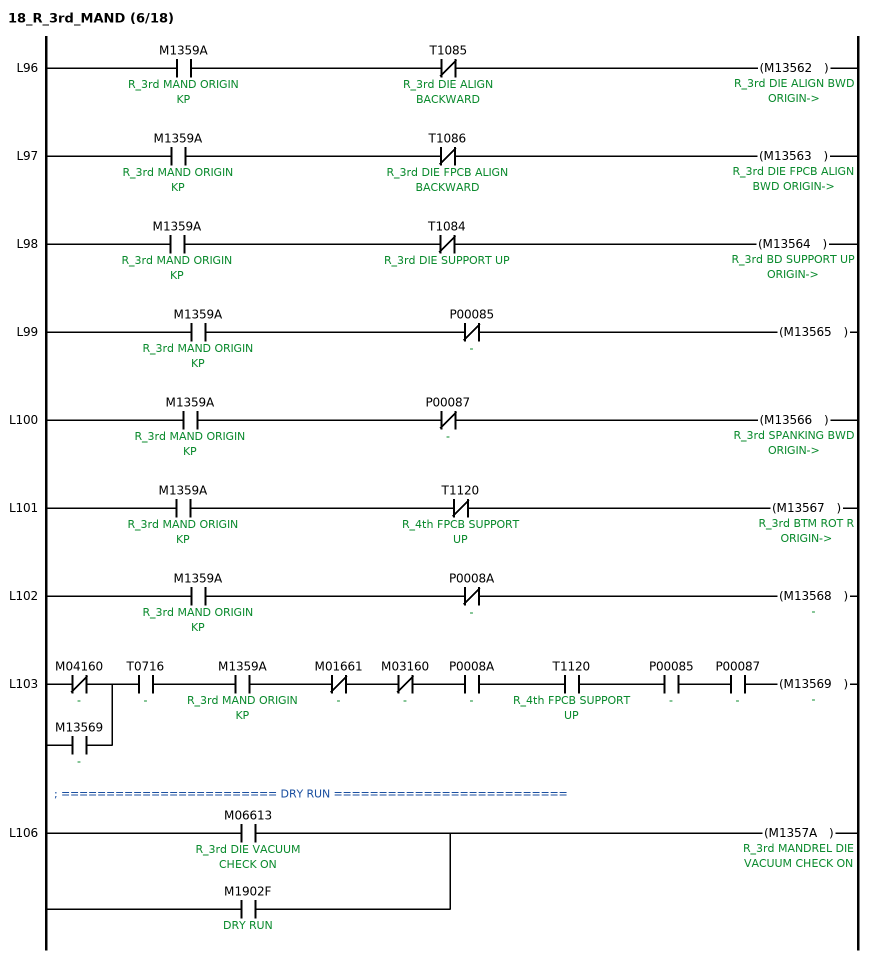
; L96
LOAD      M1359A	// R_3rd MAND ORIGIN KP
AND NOT   T1085	// R_3rd DIE ALIGN BACKWARD
OUT       M13562	// R_3rd DIE ALIGN BWD ORIGIN->
; L97
LOAD      M1359A	// R_3rd MAND ORIGIN KP
AND NOT   T1086	// R_3rd DIE FPCB ALIGN BACKWARD
OUT       M13563	// R_3rd DIE FPCB ALIGN BWD ORIGIN->
; L98
LOAD      M1359A	// R_3rd MAND ORIGIN KP
AND NOT   T1084	// R_3rd DIE SUPPORT UP
OUT       M13564	// R_3rd BD SUPPORT UP ORIGIN->
; L99
LOAD      M1359A	// R_3rd MAND ORIGIN KP
AND NOT   P00085	// -
OUT       M13565
; L100
LOAD      M1359A	// R_3rd MAND ORIGIN KP
AND NOT   P00087	// -
OUT       M13566	// R_3rd SPANKING BWD ORIGIN->
; L101
LOAD      M1359A	// R_3rd MAND ORIGIN KP
AND NOT   T1120	// R_4th FPCB SUPPORT UP
OUT       M13567	// R_3rd BTM ROT R ORIGIN->
; L102
LOAD      M1359A	// R_3rd MAND ORIGIN KP
AND NOT   P0008A	// -
OUT       M13568	// -
; L103
LOAD NOT  M04160	// -
OR        M13569	// -
AND       T0716	// -
AND       M1359A	// R_3rd MAND ORIGIN KP
AND NOT   M01661	// -
AND NOT   M03160	// -
AND       P0008A	// -
AND       T1120	// R_4th FPCB SUPPORT UP
AND       P00085	// -
AND       P00087	// -
OUT       M13569	// -
// ======================== DRY RUN ==========================
; L106
LOAD      M06613	// R_3rd DIE VACUUM CHECK ON
OR        M1902F	// DRY RUN
OUT       M1357A	// R_3rd MANDREL DIE VACUUM CHECK ON

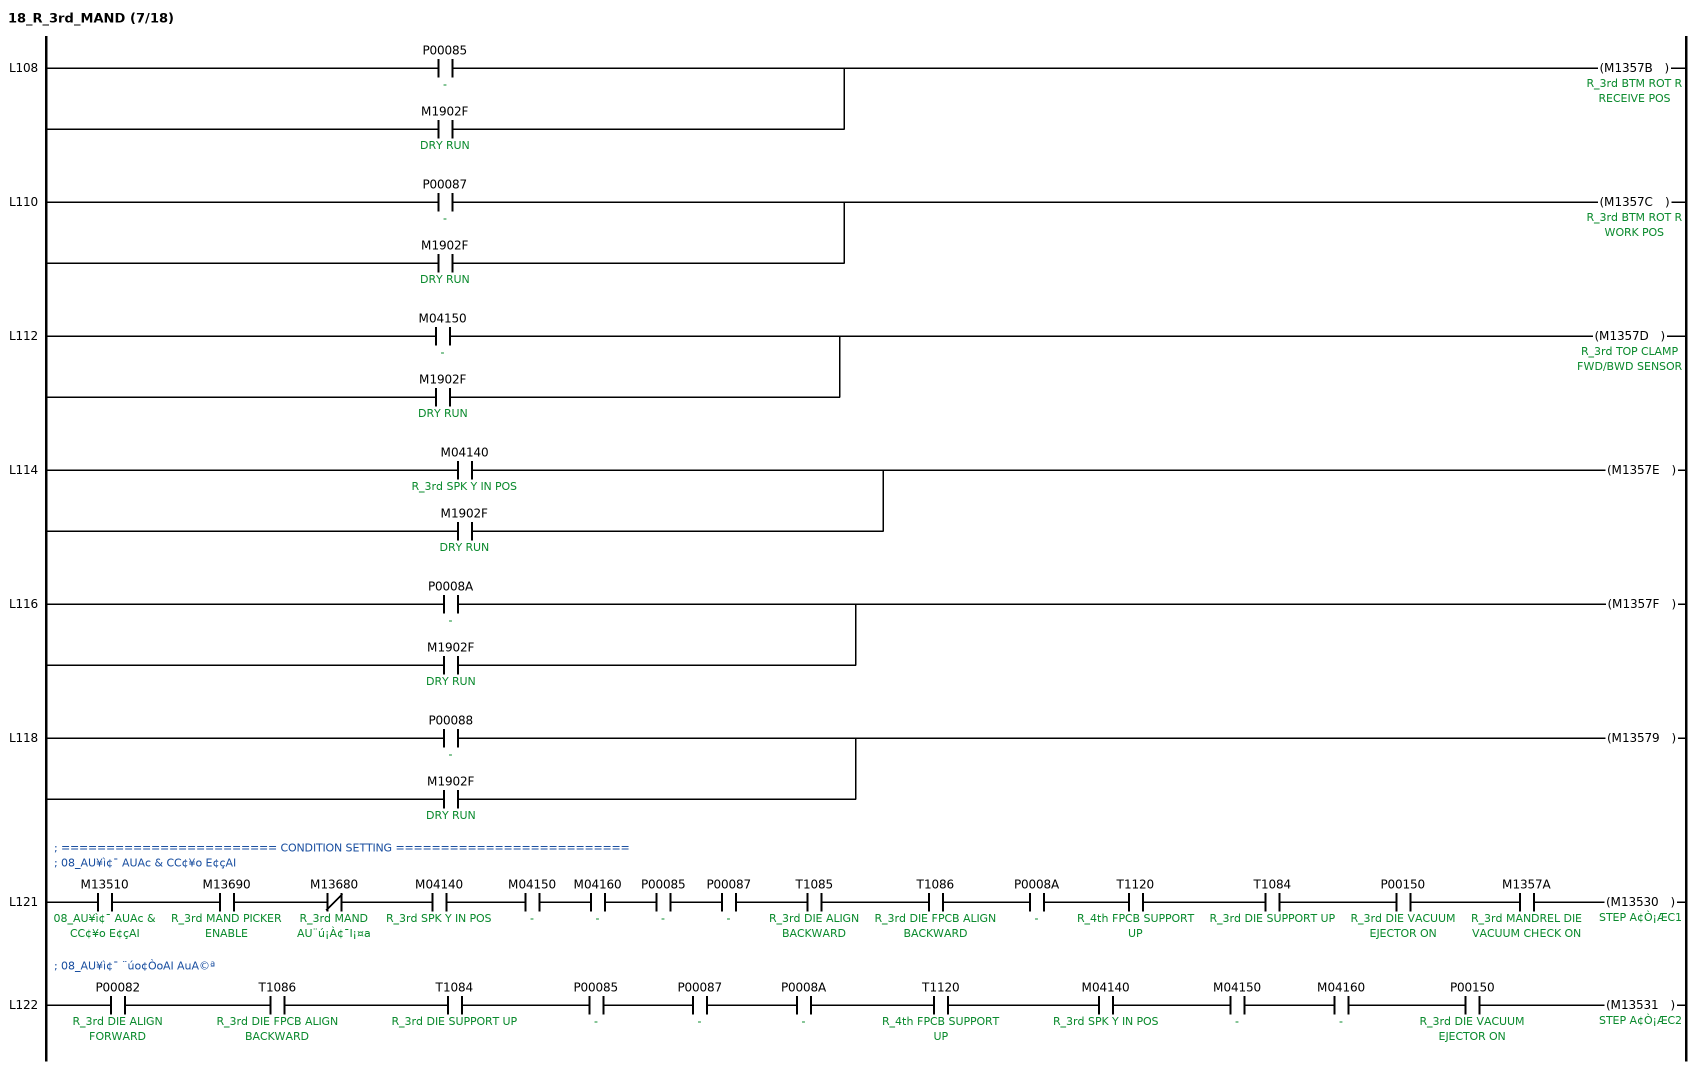
; L108
LOAD      P00085	// -
OR        M1902F	// DRY RUN
OUT       M1357B	// R_3rd BTM ROT R RECEIVE POS
; L110
LOAD      P00087	// -
OR        M1902F	// DRY RUN
OUT       M1357C	// R_3rd BTM ROT R WORK POS
; L112
LOAD      M04150	// -
OR        M1902F	// DRY RUN
OUT       M1357D	// R_3rd TOP CLAMP FWD/BWD SENSOR
; L114
LOAD      M04140	// R_3rd SPK Y IN POS
OR        M1902F	// DRY RUN
OUT       M1357E
; L116
LOAD      P0008A	// -
OR        M1902F	// DRY RUN
OUT       M1357F
; L118
LOAD      P00088	// -
OR        M1902F	// DRY RUN
OUT       M13579
// ======================== CONDITION SETTING ==========================
; L121
LOAD      M13510	// 08_AU¥ì¢¯ AUAc & CC¢¥o E¢çAI
AND       M13690	// R_3rd MAND PICKER ENABLE
AND NOT   M13680	// R_3rd MAND AU¨ú¡À¢¯I¡¤a
AND       M04140	// R_3rd SPK Y IN POS
AND       M04150	// -
AND       M04160	// -
AND       P00085	// -
AND       P00087	// -
AND       T1085	// R_3rd DIE ALIGN BACKWARD
AND       T1086	// R_3rd DIE FPCB ALIGN BACKWARD
AND       P0008A	// -
AND       T1120	// R_4th FPCB SUPPORT UP
AND       T1084	// R_3rd DIE SUPPORT UP
AND       P00150	// R_3rd DIE VACUUM EJECTOR ON
AND       M1357A	// R_3rd MANDREL DIE VACUUM CHECK ON
OUT       M13530	// STEP A¢Ò¡ÆC1
// output comment: 08_AU¥ì¢¯ AUAc & CC¢¥o E¢çAI
; L122
LOAD      P00082	// R_3rd DIE ALIGN FORWARD
AND       T1086	// R_3rd DIE FPCB ALIGN BACKWARD
AND       T1084	// R_3rd DIE SUPPORT UP
AND       P00085	// -
AND       P00087	// -
AND       P0008A	// -
AND       T1120	// R_4th FPCB SUPPORT UP
AND       M04140	// R_3rd SPK Y IN POS
AND       M04150	// -
AND       M04160	// -
AND       P00150	// R_3rd DIE VACUUM EJECTOR ON
OUT       M13531	// STEP A¢Ò¡ÆC2
// output comment: 08_AU¥ì¢¯ ¨úo¢ÒoAI AuA©ª

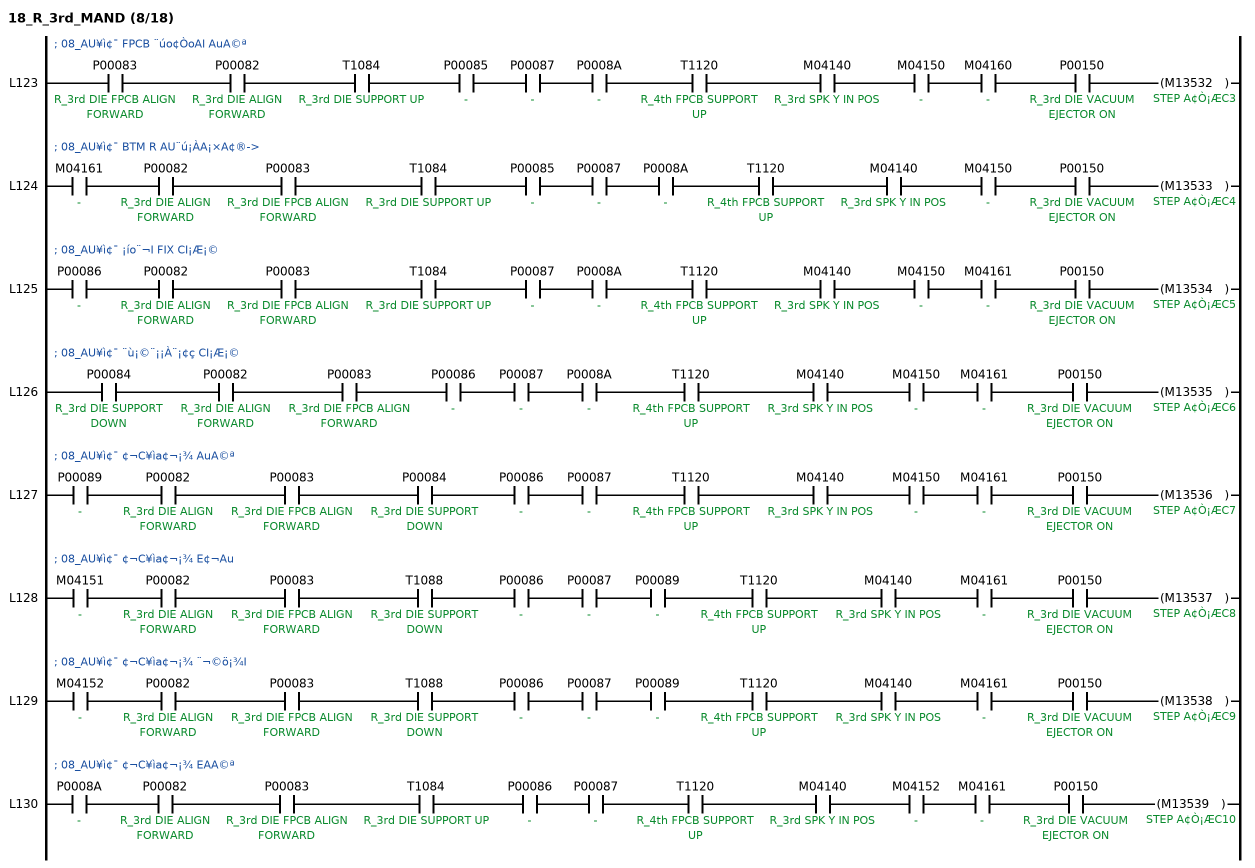
; L123
LOAD      P00083	// R_3rd DIE FPCB ALIGN FORWARD
AND       P00082	// R_3rd DIE ALIGN FORWARD
AND       T1084	// R_3rd DIE SUPPORT UP
AND       P00085	// -
AND       P00087	// -
AND       P0008A	// -
AND       T1120	// R_4th FPCB SUPPORT UP
AND       M04140	// R_3rd SPK Y IN POS
AND       M04150	// -
AND       M04160	// -
AND       P00150	// R_3rd DIE VACUUM EJECTOR ON
OUT       M13532	// STEP A¢Ò¡ÆC3
// output comment: 08_AU¥ì¢¯ FPCB ¨úo¢ÒoAI AuA©ª
; L124
LOAD      M04161	// -
AND       P00082	// R_3rd DIE ALIGN FORWARD
AND       P00083	// R_3rd DIE FPCB ALIGN FORWARD
AND       T1084	// R_3rd DIE SUPPORT UP
AND       P00085	// -
AND       P00087	// -
AND       P0008A	// -
AND       T1120	// R_4th FPCB SUPPORT UP
AND       M04140	// R_3rd SPK Y IN POS
AND       M04150	// -
AND       P00150	// R_3rd DIE VACUUM EJECTOR ON
OUT       M13533	// STEP A¢Ò¡ÆC4
// output comment: 08_AU¥ì¢¯ BTM R AU¨ú¡ÀA¡×A¢®->
; L125
LOAD      P00086	// -
AND       P00082	// R_3rd DIE ALIGN FORWARD
AND       P00083	// R_3rd DIE FPCB ALIGN FORWARD
AND       T1084	// R_3rd DIE SUPPORT UP
AND       P00087	// -
AND       P0008A	// -
AND       T1120	// R_4th FPCB SUPPORT UP
AND       M04140	// R_3rd SPK Y IN POS
AND       M04150	// -
AND       M04161	// -
AND       P00150	// R_3rd DIE VACUUM EJECTOR ON
OUT       M13534	// STEP A¢Ò¡ÆC5
// output comment: 08_AU¥ì¢¯ ¡ío¨¬I FIX CI¡Æ¡©
; L126
LOAD      P00084	// R_3rd DIE SUPPORT DOWN
AND       P00082	// R_3rd DIE ALIGN FORWARD
AND       P00083	// R_3rd DIE FPCB ALIGN FORWARD
AND       P00086	// -
AND       P00087	// -
AND       P0008A	// -
AND       T1120	// R_4th FPCB SUPPORT UP
AND       M04140	// R_3rd SPK Y IN POS
AND       M04150	// -
AND       M04161	// -
AND       P00150	// R_3rd DIE VACUUM EJECTOR ON
OUT       M13535	// STEP A¢Ò¡ÆC6
// output comment: 08_AU¥ì¢¯ ¨ù¡©¨¡¡À¨¡¢ç CI¡Æ¡©
; L127
LOAD      P00089	// -
AND       P00082	// R_3rd DIE ALIGN FORWARD
AND       P00083	// R_3rd DIE FPCB ALIGN FORWARD
AND       P00084	// R_3rd DIE SUPPORT DOWN
AND       P00086	// -
AND       P00087	// -
AND       T1120	// R_4th FPCB SUPPORT UP
AND       M04140	// R_3rd SPK Y IN POS
AND       M04150	// -
AND       M04161	// -
AND       P00150	// R_3rd DIE VACUUM EJECTOR ON
OUT       M13536	// STEP A¢Ò¡ÆC7
// output comment: 08_AU¥ì¢¯ ¢¬C¥ìa¢¬¡¾ AuA©ª
; L128
LOAD      M04151	// -
AND       P00082	// R_3rd DIE ALIGN FORWARD
AND       P00083	// R_3rd DIE FPCB ALIGN FORWARD
AND       T1088	// R_3rd DIE SUPPORT DOWN
AND       P00086	// -
AND       P00087	// -
AND       P00089	// -
AND       T1120	// R_4th FPCB SUPPORT UP
AND       M04140	// R_3rd SPK Y IN POS
AND       M04161	// -
AND       P00150	// R_3rd DIE VACUUM EJECTOR ON
OUT       M13537	// STEP A¢Ò¡ÆC8
// output comment: 08_AU¥ì¢¯ ¢¬C¥ìa¢¬¡¾ E¢¬Au
; L129
LOAD      M04152	// -
AND       P00082	// R_3rd DIE ALIGN FORWARD
AND       P00083	// R_3rd DIE FPCB ALIGN FORWARD
AND       T1088	// R_3rd DIE SUPPORT DOWN
AND       P00086	// -
AND       P00087	// -
AND       P00089	// -
AND       T1120	// R_4th FPCB SUPPORT UP
AND       M04140	// R_3rd SPK Y IN POS
AND       M04161	// -
AND       P00150	// R_3rd DIE VACUUM EJECTOR ON
OUT       M13538	// STEP A¢Ò¡ÆC9
// output comment: 08_AU¥ì¢¯ ¢¬C¥ìa¢¬¡¾ ¨¬©ö¡¾I
; L130
LOAD      P0008A	// -
AND       P00082	// R_3rd DIE ALIGN FORWARD
AND       P00083	// R_3rd DIE FPCB ALIGN FORWARD
AND       T1084	// R_3rd DIE SUPPORT UP
AND       P00086	// -
AND       P00087	// -
AND       T1120	// R_4th FPCB SUPPORT UP
AND       M04140	// R_3rd SPK Y IN POS
AND       M04152	// -
AND       M04161	// -
AND       P00150	// R_3rd DIE VACUUM EJECTOR ON
OUT       M13539	// STEP A¢Ò¡ÆC10
// output comment: 08_AU¥ì¢¯ ¢¬C¥ìa¢¬¡¾ EAA©ª

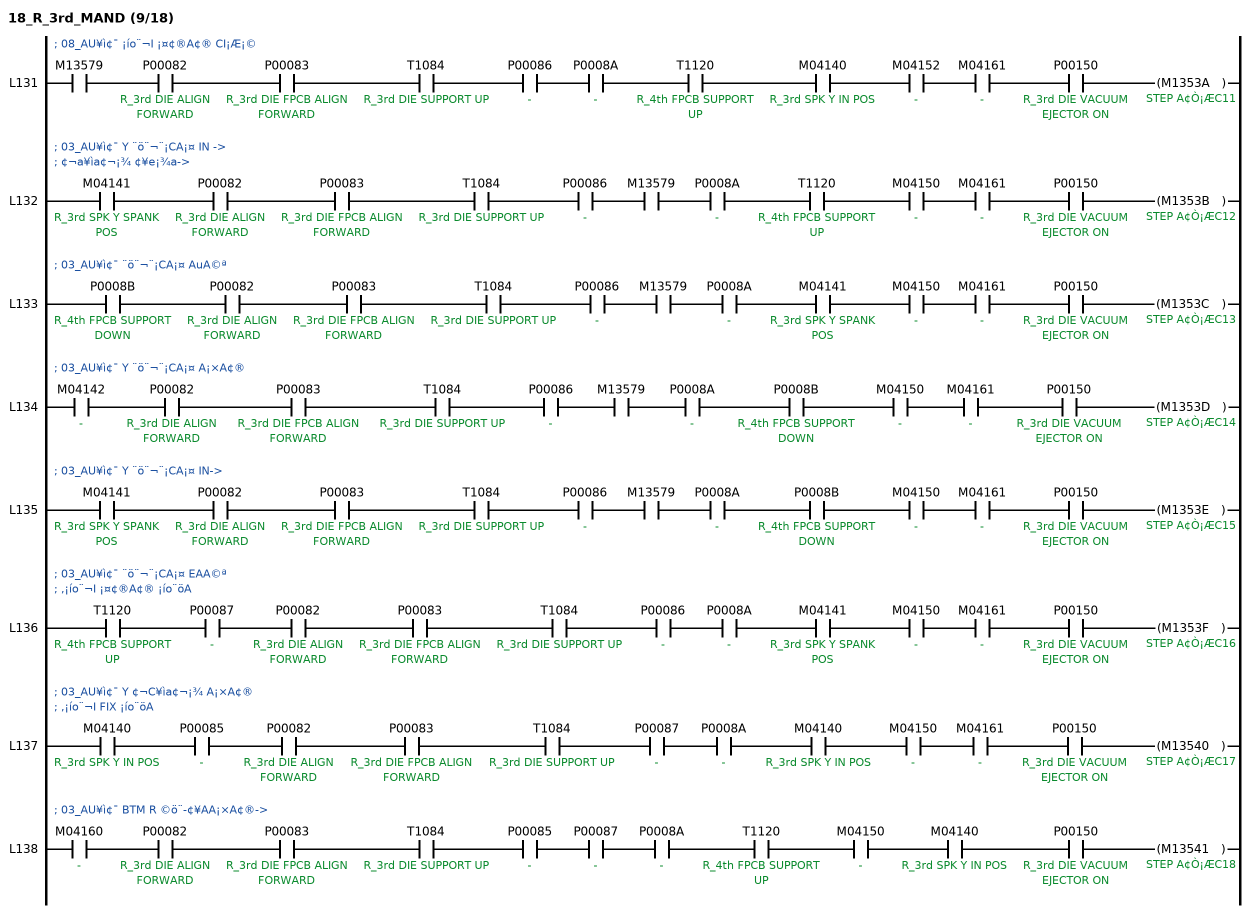
; L131
LOAD      M13579
AND       P00082	// R_3rd DIE ALIGN FORWARD
AND       P00083	// R_3rd DIE FPCB ALIGN FORWARD
AND       T1084	// R_3rd DIE SUPPORT UP
AND       P00086	// -
AND       P0008A	// -
AND       T1120	// R_4th FPCB SUPPORT UP
AND       M04140	// R_3rd SPK Y IN POS
AND       M04152	// -
AND       M04161	// -
AND       P00150	// R_3rd DIE VACUUM EJECTOR ON
OUT       M1353A	// STEP A¢Ò¡ÆC11
// output comment: 08_AU¥ì¢¯ ¡ío¨¬I ¡¤¢®A¢® CI¡Æ¡©
; L132
LOAD      M04141	// R_3rd SPK Y SPANK POS
AND       P00082	// R_3rd DIE ALIGN FORWARD
AND       P00083	// R_3rd DIE FPCB ALIGN FORWARD
AND       T1084	// R_3rd DIE SUPPORT UP
AND       P00086	// -
AND       M13579
AND       P0008A	// -
AND       T1120	// R_4th FPCB SUPPORT UP
AND       M04150	// -
AND       M04161	// -
AND       P00150	// R_3rd DIE VACUUM EJECTOR ON
OUT       M1353B	// STEP A¢Ò¡ÆC12
// output comment: 03_AU¥ì¢¯ Y ¨ö¨¬¨¡CA¡¤ IN -> ¢¬a¥ìa¢¬¡¾ ¢¥e¡¾a->
; L133
LOAD      P0008B	// R_4th FPCB SUPPORT DOWN
AND       P00082	// R_3rd DIE ALIGN FORWARD
AND       P00083	// R_3rd DIE FPCB ALIGN FORWARD
AND       T1084	// R_3rd DIE SUPPORT UP
AND       P00086	// -
AND       M13579
AND       P0008A	// -
AND       M04141	// R_3rd SPK Y SPANK POS
AND       M04150	// -
AND       M04161	// -
AND       P00150	// R_3rd DIE VACUUM EJECTOR ON
OUT       M1353C	// STEP A¢Ò¡ÆC13
// output comment: 03_AU¥ì¢¯ ¨ö¨¬¨¡CA¡¤ AuA©ª
; L134
LOAD      M04142	// -
AND       P00082	// R_3rd DIE ALIGN FORWARD
AND       P00083	// R_3rd DIE FPCB ALIGN FORWARD
AND       T1084	// R_3rd DIE SUPPORT UP
AND       P00086	// -
AND       M13579
AND       P0008A	// -
AND       P0008B	// R_4th FPCB SUPPORT DOWN
AND       M04150	// -
AND       M04161	// -
AND       P00150	// R_3rd DIE VACUUM EJECTOR ON
OUT       M1353D	// STEP A¢Ò¡ÆC14
// output comment: 03_AU¥ì¢¯ Y ¨ö¨¬¨¡CA¡¤ A¡×A¢®
; L135
LOAD      M04141	// R_3rd SPK Y SPANK POS
AND       P00082	// R_3rd DIE ALIGN FORWARD
AND       P00083	// R_3rd DIE FPCB ALIGN FORWARD
AND       T1084	// R_3rd DIE SUPPORT UP
AND       P00086	// -
AND       M13579
AND       P0008A	// -
AND       P0008B	// R_4th FPCB SUPPORT DOWN
AND       M04150	// -
AND       M04161	// -
AND       P00150	// R_3rd DIE VACUUM EJECTOR ON
OUT       M1353E	// STEP A¢Ò¡ÆC15
// output comment: 03_AU¥ì¢¯ Y ¨ö¨¬¨¡CA¡¤ IN->
; L136
LOAD      T1120	// R_4th FPCB SUPPORT UP
AND       P00087	// -
AND       P00082	// R_3rd DIE ALIGN FORWARD
AND       P00083	// R_3rd DIE FPCB ALIGN FORWARD
AND       T1084	// R_3rd DIE SUPPORT UP
AND       P00086	// -
AND       P0008A	// -
AND       M04141	// R_3rd SPK Y SPANK POS
AND       M04150	// -
AND       M04161	// -
AND       P00150	// R_3rd DIE VACUUM EJECTOR ON
OUT       M1353F	// STEP A¢Ò¡ÆC16
// output comment: 03_AU¥ì¢¯ ¨ö¨¬¨¡CA¡¤ EAA©ª ,¡ío¨¬I ¡¤¢®A¢® ¡ío¨öA
; L137
LOAD      M04140	// R_3rd SPK Y IN POS
AND       P00085	// -
AND       P00082	// R_3rd DIE ALIGN FORWARD
AND       P00083	// R_3rd DIE FPCB ALIGN FORWARD
AND       T1084	// R_3rd DIE SUPPORT UP
AND       P00087	// -
AND       P0008A	// -
AND       M04140	// R_3rd SPK Y IN POS
AND       M04150	// -
AND       M04161	// -
AND       P00150	// R_3rd DIE VACUUM EJECTOR ON
OUT       M13540	// STEP A¢Ò¡ÆC17
// output comment: 03_AU¥ì¢¯ Y ¢¬C¥ìa¢¬¡¾ A¡×A¢® ,¡ío¨¬I FIX ¡ío¨öA
; L138
LOAD      M04160	// -
AND       P00082	// R_3rd DIE ALIGN FORWARD
AND       P00083	// R_3rd DIE FPCB ALIGN FORWARD
AND       T1084	// R_3rd DIE SUPPORT UP
AND       P00085	// -
AND       P00087	// -
AND       P0008A	// -
AND       T1120	// R_4th FPCB SUPPORT UP
AND       M04150	// -
AND       M04140	// R_3rd SPK Y IN POS
AND       P00150	// R_3rd DIE VACUUM EJECTOR ON
OUT       M13541	// STEP A¢Ò¡ÆC18
// output comment: 03_AU¥ì¢¯ BTM R ©ö¨­¢¥AA¡×A¢®->

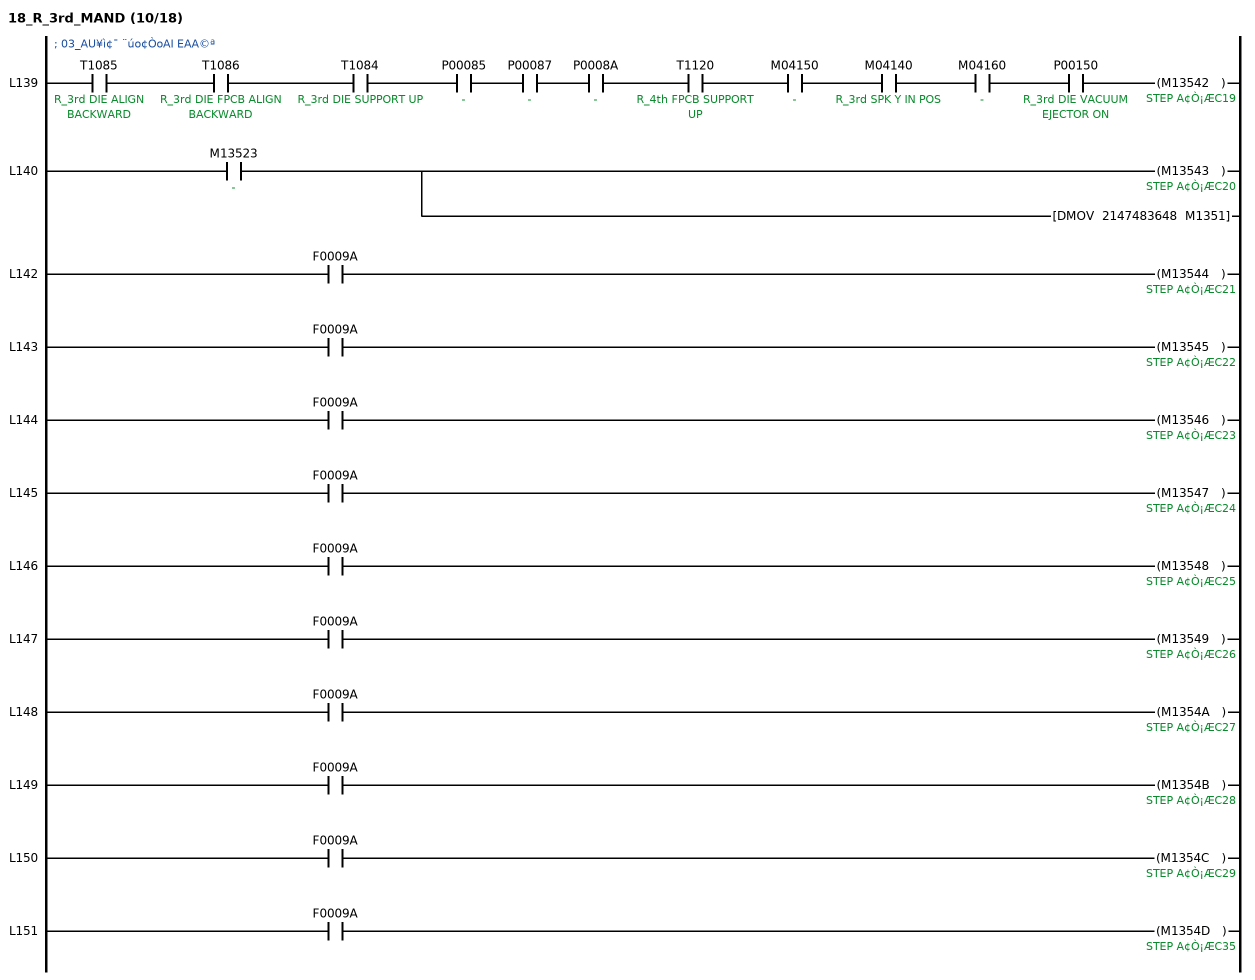
; L139
LOAD      T1085	// R_3rd DIE ALIGN BACKWARD
AND       T1086	// R_3rd DIE FPCB ALIGN BACKWARD
AND       T1084	// R_3rd DIE SUPPORT UP
AND       P00085	// -
AND       P00087	// -
AND       P0008A	// -
AND       T1120	// R_4th FPCB SUPPORT UP
AND       M04150	// -
AND       M04140	// R_3rd SPK Y IN POS
AND       M04160	// -
AND       P00150	// R_3rd DIE VACUUM EJECTOR ON
OUT       M13542	// STEP A¢Ò¡ÆC19
// output comment: 03_AU¥ì¢¯ ¨úo¢ÒoAI EAA©ª
; L140
LOAD      M13523	// -
OUT       M13543	// STEP A¢Ò¡ÆC20
DMOV      2147483648 M1351
; L142
LOAD      F0009A
OUT       M13544	// STEP A¢Ò¡ÆC21
; L143
LOAD      F0009A
OUT       M13545	// STEP A¢Ò¡ÆC22
; L144
LOAD      F0009A
OUT       M13546	// STEP A¢Ò¡ÆC23
; L145
LOAD      F0009A
OUT       M13547	// STEP A¢Ò¡ÆC24
; L146
LOAD      F0009A
OUT       M13548	// STEP A¢Ò¡ÆC25
; L147
LOAD      F0009A
OUT       M13549	// STEP A¢Ò¡ÆC26
; L148
LOAD      F0009A
OUT       M1354A	// STEP A¢Ò¡ÆC27
; L149
LOAD      F0009A
OUT       M1354B	// STEP A¢Ò¡ÆC28
; L150
LOAD      F0009A
OUT       M1354C	// STEP A¢Ò¡ÆC29
; L151
LOAD      F0009A
OUT       M1354D	// STEP A¢Ò¡ÆC35

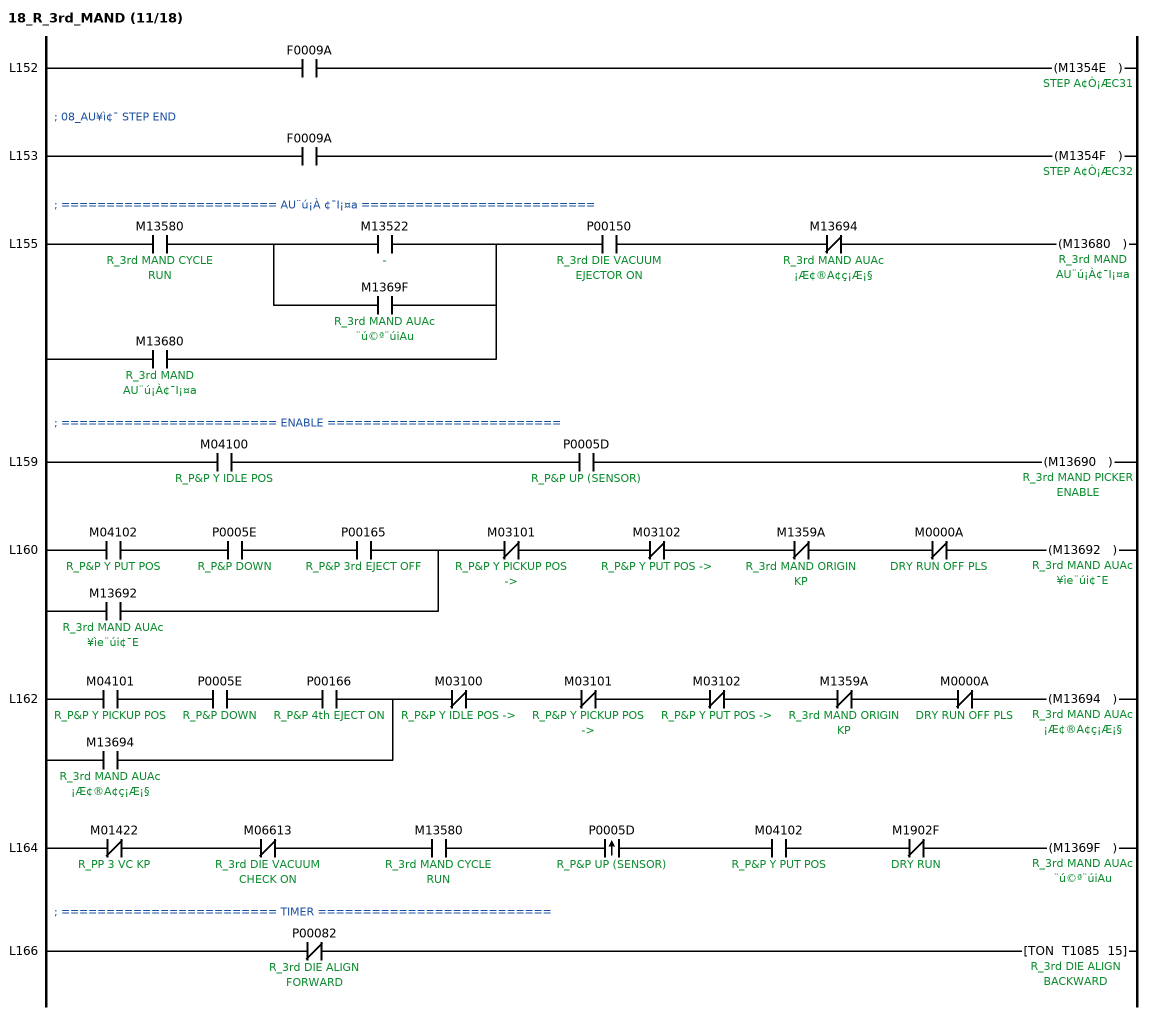
; L152
LOAD      F0009A
OUT       M1354E	// STEP A¢Ò¡ÆC31
; L153
LOAD      F0009A
OUT       M1354F	// STEP A¢Ò¡ÆC32
// output comment: 08_AU¥ì¢¯ STEP END
// ======================== AU¨ú¡À ¢¯I¡¤a ==========================
; L155
LOAD      M13580	// R_3rd MAND CYCLE RUN
LOAD      M13522	// -
OR        M1369F	// R_3rd MAND AUAc ¨ú©ª¨úiAu
AND LOAD
OR        M13680	// R_3rd MAND AU¨ú¡À¢¯I¡¤a
AND       P00150	// R_3rd DIE VACUUM EJECTOR ON
AND NOT   M13694	// R_3rd MAND AUAc ¡Æ¢®A¢ç¡Æ¡§
OUT       M13680	// R_3rd MAND AU¨ú¡À¢¯I¡¤a
// ======================== ENABLE ==========================
; L159
LOAD      M04100	// R_P&P Y IDLE POS
AND       P0005D	// R_P&P UP (SENSOR)
OUT       M13690	// R_3rd MAND PICKER ENABLE
; L160
LOAD      M04102	// R_P&P Y PUT POS
AND       P0005E	// R_P&P DOWN
AND       P00165	// R_P&P 3rd EJECT OFF
OR        M13692	// R_3rd MAND AUAc ¥ìe¨úi¢¯E
AND NOT   M03101	// R_P&P Y PICKUP POS ->
AND NOT   M03102	// R_P&P Y PUT POS ->
AND NOT   M1359A	// R_3rd MAND ORIGIN KP
AND NOT   M0000A	// DRY RUN OFF PLS
OUT       M13692	// R_3rd MAND AUAc ¥ìe¨úi¢¯E
; L162
LOAD      M04101	// R_P&P Y PICKUP POS
AND       P0005E	// R_P&P DOWN
AND       P00166	// R_P&P 4th EJECT ON
OR        M13694	// R_3rd MAND AUAc ¡Æ¢®A¢ç¡Æ¡§
AND NOT   M03100	// R_P&P Y IDLE POS ->
AND NOT   M03101	// R_P&P Y PICKUP POS ->
AND NOT   M03102	// R_P&P Y PUT POS ->
AND NOT   M1359A	// R_3rd MAND ORIGIN KP
AND NOT   M0000A	// DRY RUN OFF PLS
OUT       M13694	// R_3rd MAND AUAc ¡Æ¢®A¢ç¡Æ¡§
; L164
LOAD NOT  M01422	// R_PP 3 VC KP
AND NOT   M06613	// R_3rd DIE VACUUM CHECK ON
AND       M13580	// R_3rd MAND CYCLE RUN
ANDP      P0005D	// R_P&P UP (SENSOR)
AND       M04102	// R_P&P Y PUT POS
AND NOT   M1902F	// DRY RUN
OUT       M1369F	// R_3rd MAND AUAc ¨ú©ª¨úiAu
// ======================== TIMER ==========================
; L166
LOAD NOT  P00082	// R_3rd DIE ALIGN FORWARD
TON       T1085 15	// R_3rd DIE ALIGN BACKWARD

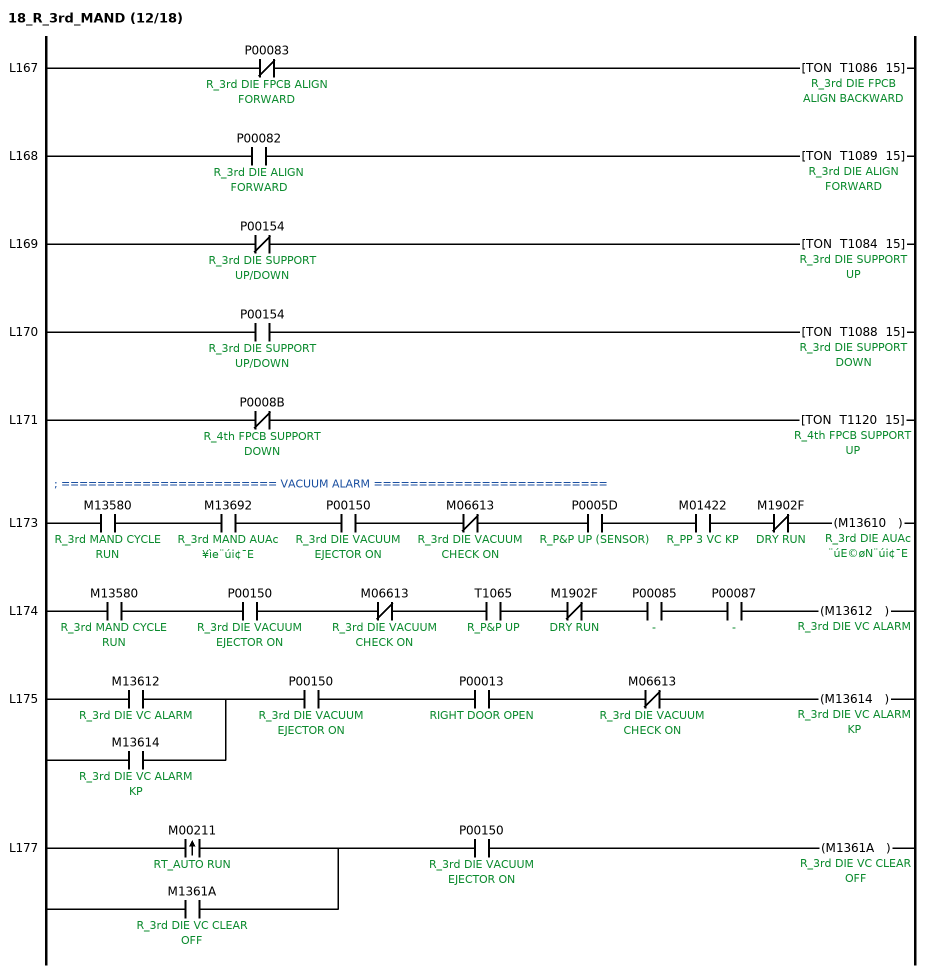
; L167
LOAD NOT  P00083	// R_3rd DIE FPCB ALIGN FORWARD
TON       T1086 15	// R_3rd DIE FPCB ALIGN BACKWARD
; L168
LOAD      P00082	// R_3rd DIE ALIGN FORWARD
TON       T1089 15	// R_3rd DIE ALIGN FORWARD
; L169
LOAD NOT  P00154	// R_3rd DIE SUPPORT UP/DOWN
TON       T1084 15	// R_3rd DIE SUPPORT UP
; L170
LOAD      P00154	// R_3rd DIE SUPPORT UP/DOWN
TON       T1088 15	// R_3rd DIE SUPPORT DOWN
; L171
LOAD NOT  P0008B	// R_4th FPCB SUPPORT DOWN
TON       T1120 15	// R_4th FPCB SUPPORT UP
// ======================== VACUUM ALARM ==========================
; L173
LOAD      M13580	// R_3rd MAND CYCLE RUN
AND       M13692	// R_3rd MAND AUAc ¥ìe¨úi¢¯E
AND       P00150	// R_3rd DIE VACUUM EJECTOR ON
AND NOT   M06613	// R_3rd DIE VACUUM CHECK ON
AND       P0005D	// R_P&P UP (SENSOR)
AND       M01422	// R_PP 3 VC KP
AND NOT   M1902F	// DRY RUN
OUT       M13610	// R_3rd DIE AUAc ¨úE©øN¨úi¢¯E
; L174
LOAD      M13580	// R_3rd MAND CYCLE RUN
AND       P00150	// R_3rd DIE VACUUM EJECTOR ON
AND NOT   M06613	// R_3rd DIE VACUUM CHECK ON
AND       T1065	// R_P&P UP
AND NOT   M1902F	// DRY RUN
AND       P00085	// -
AND       P00087	// -
OUT       M13612	// R_3rd DIE VC ALARM
; L175
LOAD      M13612	// R_3rd DIE VC ALARM
OR        M13614	// R_3rd DIE VC ALARM KP
AND       P00150	// R_3rd DIE VACUUM EJECTOR ON
AND       P00013	// RIGHT DOOR OPEN
AND NOT   M06613	// R_3rd DIE VACUUM CHECK ON
OUT       M13614	// R_3rd DIE VC ALARM KP
; L177
LOADP     M00211	// RT_AUTO RUN
OR        M1361A	// R_3rd DIE VC CLEAR OFF
AND       P00150	// R_3rd DIE VACUUM EJECTOR ON
OUT       M1361A	// R_3rd DIE VC CLEAR OFF

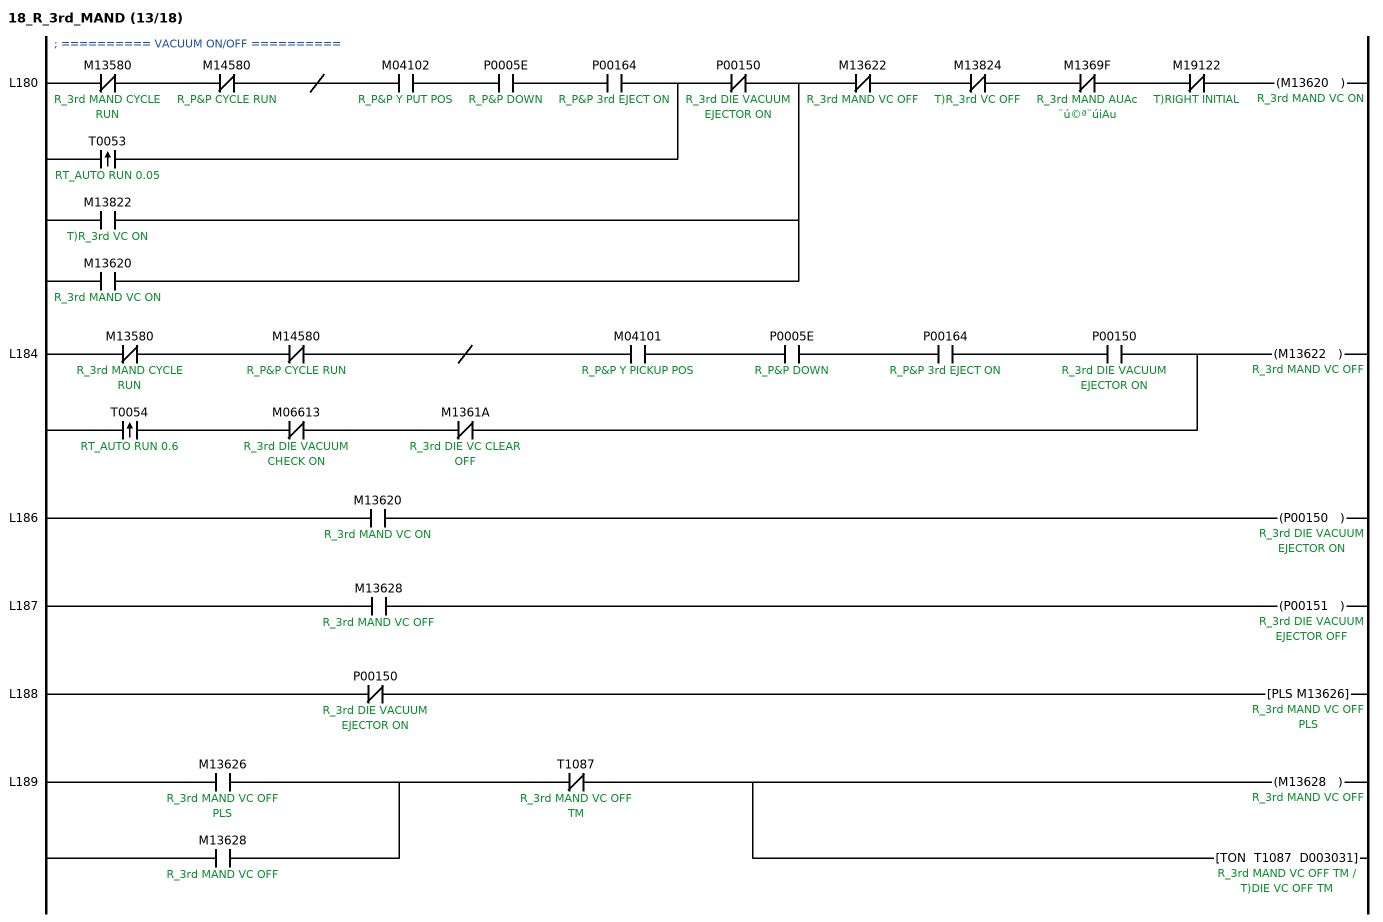
// ========== VACUUM ON/OFF ==========
; L180
LOAD NOT  M13580	// R_3rd MAND CYCLE RUN
AND NOT   M14580	// R_P&P CYCLE RUN
NOT
AND       M04102	// R_P&P Y PUT POS
AND       P0005E	// R_P&P DOWN
AND       P00164	// R_P&P 3rd EJECT ON
ORP       T0053	// RT_AUTO RUN 0.05
AND NOT   P00150	// R_3rd DIE VACUUM EJECTOR ON
OR        M13822	// T)R_3rd VC ON
OR        M13620	// R_3rd MAND VC ON
AND NOT   M13622	// R_3rd MAND VC OFF
AND NOT   M13824	// T)R_3rd VC OFF
AND NOT   M1369F	// R_3rd MAND AUAc ¨ú©ª¨úiAu
AND NOT   M19122	// T)RIGHT INITIAL
OUT       M13620	// R_3rd MAND VC ON
; L184
LOAD NOT  M13580	// R_3rd MAND CYCLE RUN
AND NOT   M14580	// R_P&P CYCLE RUN
NOT
AND       M04101	// R_P&P Y PICKUP POS
AND       P0005E	// R_P&P DOWN
AND       P00164	// R_P&P 3rd EJECT ON
AND       P00150	// R_3rd DIE VACUUM EJECTOR ON
LOADP     T0054	// RT_AUTO RUN 0.6
AND NOT   M06613	// R_3rd DIE VACUUM CHECK ON
AND NOT   M1361A	// R_3rd DIE VC CLEAR OFF
OR LOAD
OUT       M13622	// R_3rd MAND VC OFF
; L186
LOAD      M13620	// R_3rd MAND VC ON
OUT       P00150	// R_3rd DIE VACUUM EJECTOR ON
; L187
LOAD      M13628	// R_3rd MAND VC OFF
OUT       P00151	// R_3rd DIE VACUUM EJECTOR OFF
; L188
LOAD NOT  P00150	// R_3rd DIE VACUUM EJECTOR ON
OUTP      M13626	// R_3rd MAND VC OFF PLS
; L189
LOAD      M13626	// R_3rd MAND VC OFF PLS
OR        M13628	// R_3rd MAND VC OFF
AND NOT   T1087	// R_3rd MAND VC OFF TM
OUT       M13628	// R_3rd MAND VC OFF
TON       T1087 D003031	// R_3rd MAND VC OFF TM / T)DIE VC OFF TM

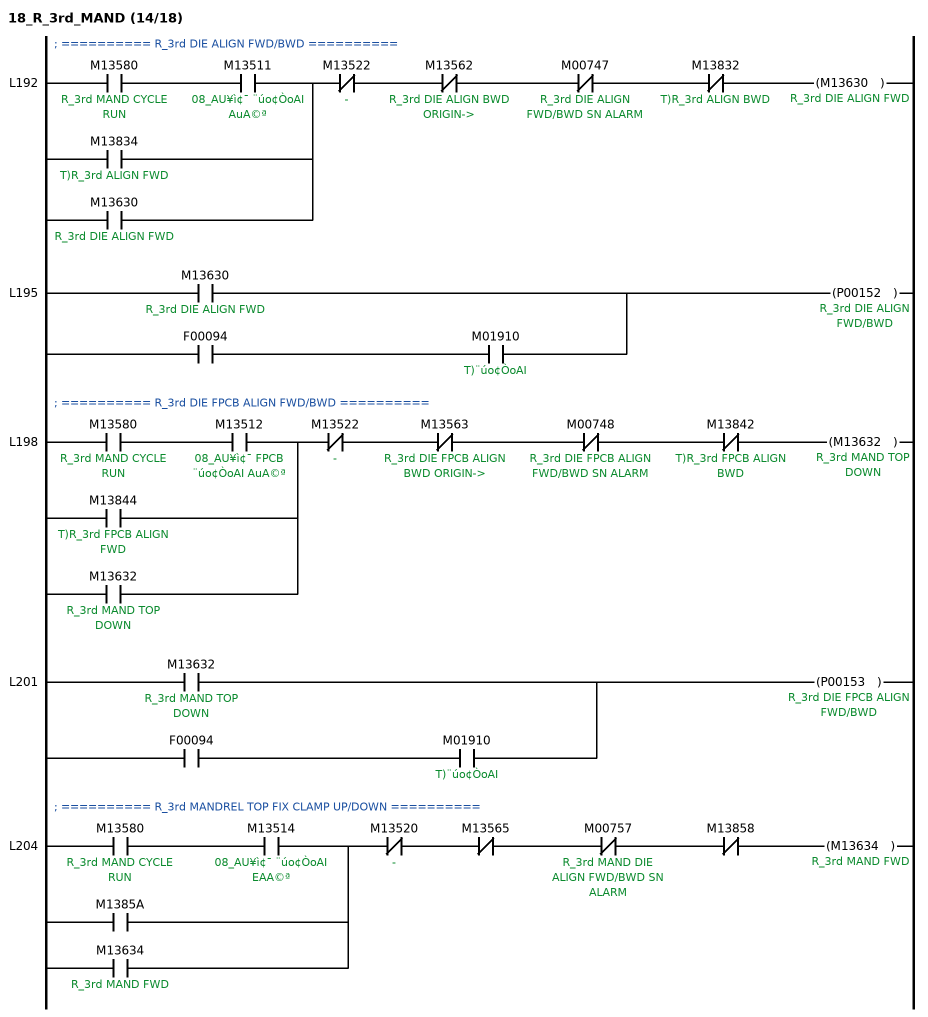
// ========== R_3rd DIE ALIGN FWD/BWD ==========
; L192
LOAD      M13580	// R_3rd MAND CYCLE RUN
AND       M13511	// 08_AU¥ì¢¯ ¨úo¢ÒoAI AuA©ª
OR        M13834	// T)R_3rd ALIGN FWD
OR        M13630	// R_3rd DIE ALIGN FWD
AND NOT   M13522	// -
AND NOT   M13562	// R_3rd DIE ALIGN BWD ORIGIN->
AND NOT   M00747	// R_3rd DIE ALIGN FWD/BWD SN ALARM
AND NOT   M13832	// T)R_3rd ALIGN BWD
OUT       M13630	// R_3rd DIE ALIGN FWD
; L195
LOAD      M13630	// R_3rd DIE ALIGN FWD
LOAD      F00094
AND       M01910	// T)¨úo¢ÒoAI
OR LOAD
OUT       P00152	// R_3rd DIE ALIGN FWD/BWD
// ========== R_3rd DIE FPCB ALIGN FWD/BWD ==========
; L198
LOAD      M13580	// R_3rd MAND CYCLE RUN
AND       M13512	// 08_AU¥ì¢¯ FPCB ¨úo¢ÒoAI AuA©ª
OR        M13844	// T)R_3rd FPCB ALIGN FWD
OR        M13632	// R_3rd MAND TOP DOWN
AND NOT   M13522	// -
AND NOT   M13563	// R_3rd DIE FPCB ALIGN BWD ORIGIN->
AND NOT   M00748	// R_3rd DIE FPCB ALIGN FWD/BWD SN ALARM
AND NOT   M13842	// T)R_3rd FPCB ALIGN BWD
OUT       M13632	// R_3rd MAND TOP DOWN
; L201
LOAD      M13632	// R_3rd MAND TOP DOWN
LOAD      F00094
AND       M01910	// T)¨úo¢ÒoAI
OR LOAD
OUT       P00153	// R_3rd DIE FPCB ALIGN FWD/BWD
// ========== R_3rd MANDREL TOP FIX CLAMP UP/DOWN ==========
; L204
LOAD      M13580	// R_3rd MAND CYCLE RUN
AND       M13514	// 08_AU¥ì¢¯ ¨úo¢ÒoAI EAA©ª
OR        M1385A
OR        M13634	// R_3rd MAND FWD
AND NOT   M13520	// -
AND NOT   M13565
AND NOT   M00757	// R_3rd MAND DIE ALIGN FWD/BWD SN ALARM
AND NOT   M13858
OUT       M13634	// R_3rd MAND FWD

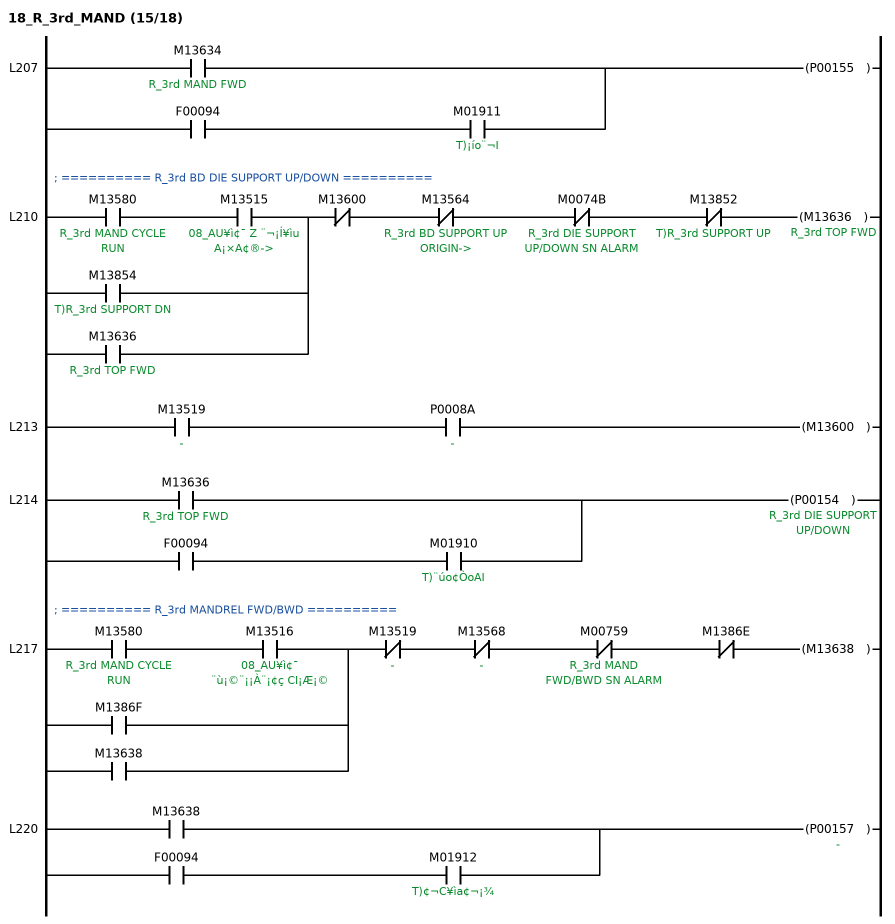
; L207
LOAD      M13634	// R_3rd MAND FWD
LOAD      F00094
AND       M01911	// T)¡ío¨¬I
OR LOAD
OUT       P00155
// ========== R_3rd BD DIE SUPPORT UP/DOWN ==========
; L210
LOAD      M13580	// R_3rd MAND CYCLE RUN
AND       M13515	// 08_AU¥ì¢¯ Z ¨¬¡Í¥ìu A¡×A¢®->
OR        M13854	// T)R_3rd SUPPORT DN
OR        M13636	// R_3rd TOP FWD
AND NOT   M13600
AND NOT   M13564	// R_3rd BD SUPPORT UP ORIGIN->
AND NOT   M0074B	// R_3rd DIE SUPPORT UP/DOWN SN ALARM
AND NOT   M13852	// T)R_3rd SUPPORT UP
OUT       M13636	// R_3rd TOP FWD
; L213
LOAD      M13519	// -
AND       P0008A	// -
OUT       M13600
; L214
LOAD      M13636	// R_3rd TOP FWD
LOAD      F00094
AND       M01910	// T)¨úo¢ÒoAI
OR LOAD
OUT       P00154	// R_3rd DIE SUPPORT UP/DOWN
// ========== R_3rd MANDREL FWD/BWD ==========
; L217
LOAD      M13580	// R_3rd MAND CYCLE RUN
AND       M13516	// 08_AU¥ì¢¯ ¨ù¡©¨¡¡À¨¡¢ç CI¡Æ¡©
OR        M1386F
OR        M13638
AND NOT   M13519	// -
AND NOT   M13568	// -
AND NOT   M00759	// R_3rd MAND FWD/BWD SN ALARM
AND NOT   M1386E
OUT       M13638
; L220
LOAD      M13638
LOAD      F00094
AND       M01912	// T)¢¬C¥ìa¢¬¡¾
OR LOAD
OUT       P00157	// -

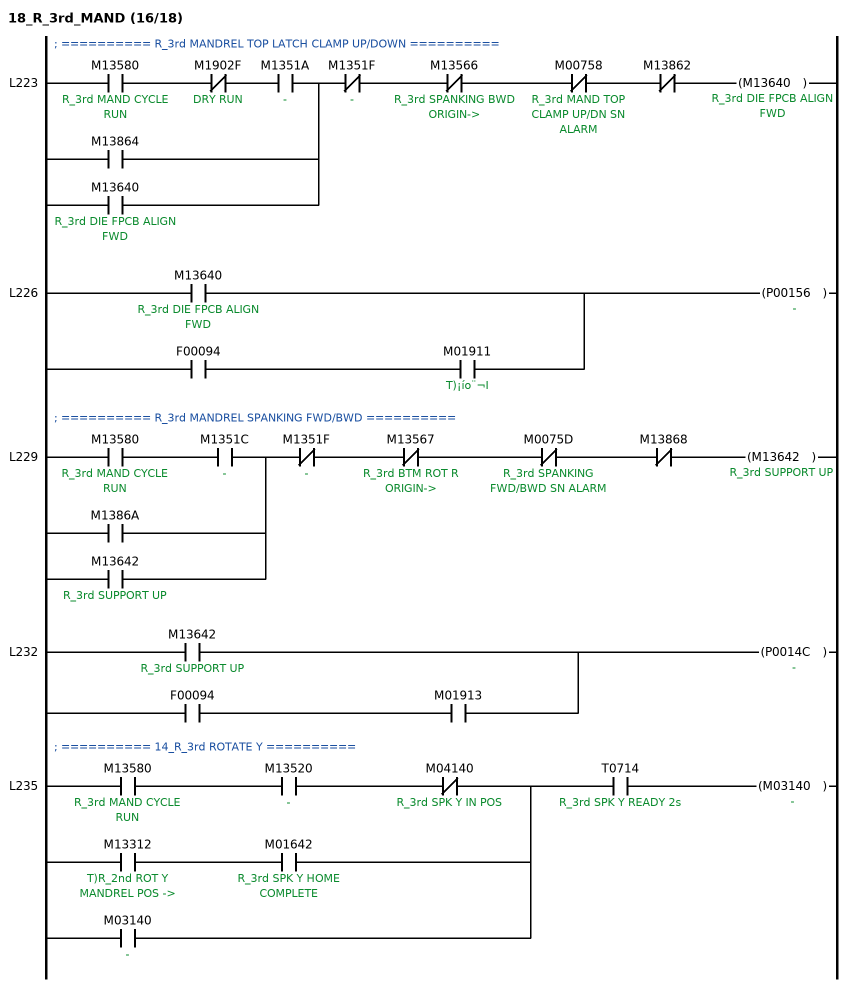
// ========== R_3rd MANDREL TOP LATCH CLAMP UP/DOWN ==========
; L223
LOAD      M13580	// R_3rd MAND CYCLE RUN
AND NOT   M1902F	// DRY RUN
AND       M1351A	// -
OR        M13864
OR        M13640	// R_3rd DIE FPCB ALIGN FWD
AND NOT   M1351F	// -
AND NOT   M13566	// R_3rd SPANKING BWD ORIGIN->
AND NOT   M00758	// R_3rd MAND TOP CLAMP UP/DN SN ALARM
AND NOT   M13862
OUT       M13640	// R_3rd DIE FPCB ALIGN FWD
; L226
LOAD      M13640	// R_3rd DIE FPCB ALIGN FWD
LOAD      F00094
AND       M01911	// T)¡ío¨¬I
OR LOAD
OUT       P00156	// -
// ========== R_3rd MANDREL SPANKING FWD/BWD ==========
; L229
LOAD      M13580	// R_3rd MAND CYCLE RUN
AND       M1351C	// -
OR        M1386A
OR        M13642	// R_3rd SUPPORT UP
AND NOT   M1351F	// -
AND NOT   M13567	// R_3rd BTM ROT R ORIGIN->
AND NOT   M0075D	// R_3rd SPANKING FWD/BWD SN ALARM
AND NOT   M13868
OUT       M13642	// R_3rd SUPPORT UP
; L232
LOAD      M13642	// R_3rd SUPPORT UP
LOAD      F00094
AND       M01913
OR LOAD
OUT       P0014C	// -
// ========== 14_R_3rd ROTATE Y ==========
; L235
LOAD      M13580	// R_3rd MAND CYCLE RUN
AND       M13520	// -
AND NOT   M04140	// R_3rd SPK Y IN POS
LOAD      M13312	// T)R_2nd ROT Y MANDREL POS ->
AND       M01642	// R_3rd SPK Y HOME COMPLETE
OR LOAD
OR        M03140	// -
AND       T0714	// R_3rd SPK Y READY 2s
OUT       M03140	// -

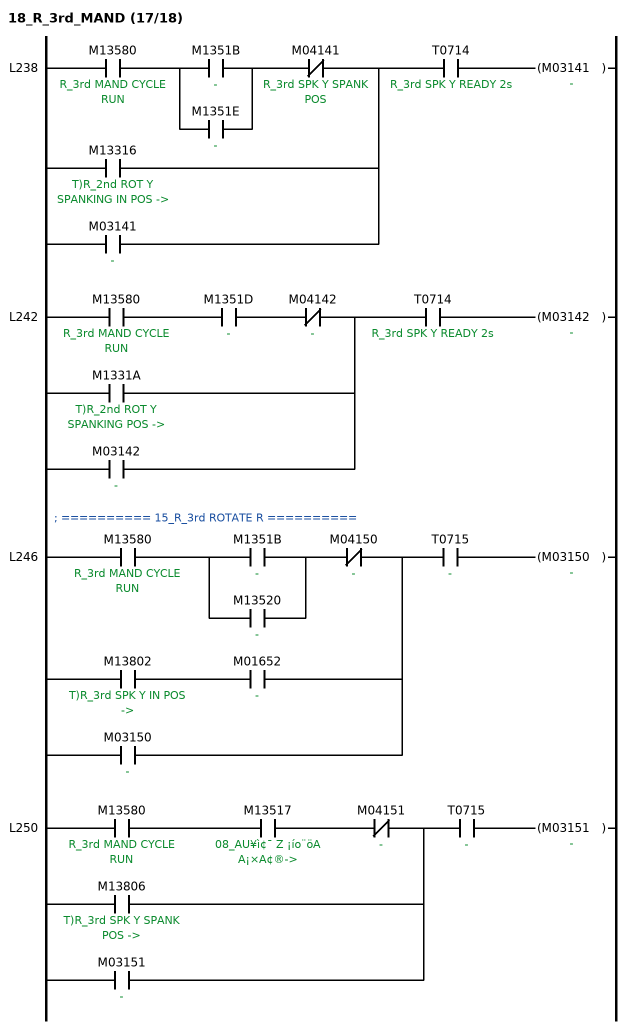
; L238
LOAD      M13580	// R_3rd MAND CYCLE RUN
LOAD      M1351B	// -
OR        M1351E	// -
AND LOAD
AND NOT   M04141	// R_3rd SPK Y SPANK POS
OR        M13316	// T)R_2nd ROT Y SPANKING IN POS ->
OR        M03141	// -
AND       T0714	// R_3rd SPK Y READY 2s
OUT       M03141	// -
; L242
LOAD      M13580	// R_3rd MAND CYCLE RUN
AND       M1351D	// -
AND NOT   M04142	// -
OR        M1331A	// T)R_2nd ROT Y SPANKING POS ->
OR        M03142	// -
AND       T0714	// R_3rd SPK Y READY 2s
OUT       M03142	// -
// ========== 15_R_3rd ROTATE R ==========
; L246
LOAD      M13580	// R_3rd MAND CYCLE RUN
LOAD      M1351B	// -
OR        M13520	// -
AND LOAD
AND NOT   M04150	// -
LOAD      M13802	// T)R_3rd SPK Y IN POS ->
AND       M01652	// -
OR LOAD
OR        M03150	// -
AND       T0715	// -
OUT       M03150	// -
; L250
LOAD      M13580	// R_3rd MAND CYCLE RUN
AND       M13517	// 08_AU¥ì¢¯ Z ¡ío¨öA A¡×A¢®->
AND NOT   M04151	// -
OR        M13806	// T)R_3rd SPK Y SPANK POS ->
OR        M03151	// -
AND       T0715	// -
OUT       M03151	// -

